# B&R Automation Studio project GroupProjectBR
Automation Studio 4.12.4.107 SP; Project that includes both HMI visualization and script of controling conveyor belt and sorting system.; technology packages: mapp 5.23.0, mappCockpit 5.23.0, mappMotion 5.23.0, mappView 5.23.0, mappVision 5.23.0

## Configuration ConfigSortingSystem

CPU , AutomationRuntime B4.93, Build 4.1.2, Safety 0.0, Vc V4.72.6

### Task classes (Cpu.sw)
```
Cyclic#1 (cycle 8000 us, tolerance 0 us):
  Auto <- Programs.Auto.prg
  Manual <- Programs.Manual.prg
  SemiAuto <- Programs.SemiAuto.prg
Cyclic#3:
  Camera <- Programs.Camera.prg
  ProgramRec <- Programs.RecipesMgmnt.prg
Cyclic#6:
  Alarms <- Programs.Alarms.prg
DataObjects: McAcpSys
NcDataObjects: McDriveLog
Binaries: McAcpDrv, udbdef, McAcpSim, mvLoader, arflatprv, TCLang, visionUnit, mCoWebSc, TCData, FWRules, arcoal, arsvcreg, SettingsVi, sysconf, Settings, iomap, asfw, Role, ashwac, gRecipeXML, Config_2, arconfig, viAppLogo, Config_1, TC, ashwd, Config, User, Config_3, viAppLogoR, viComp4, viComp1, ViApplicat, Config_5, viComp
Libraries: McBase, MpAxis, McAxis, MpBase, McAcpAx, CoTrace, AsZip, FileIO, runtime, ViBase, AsARCfg, powerlnk, MpRecipe, AsEPL, AsIO, DataObj, astime, MpAlarmX, MpServer, standard, AsHttp, asstring, MpUserX, MpFile, asieccon, aruser, arssl, sys_lib, arcert, ashw, aseth, asbrstr, asusb, MpAudit, MpReport
```

### Hardware
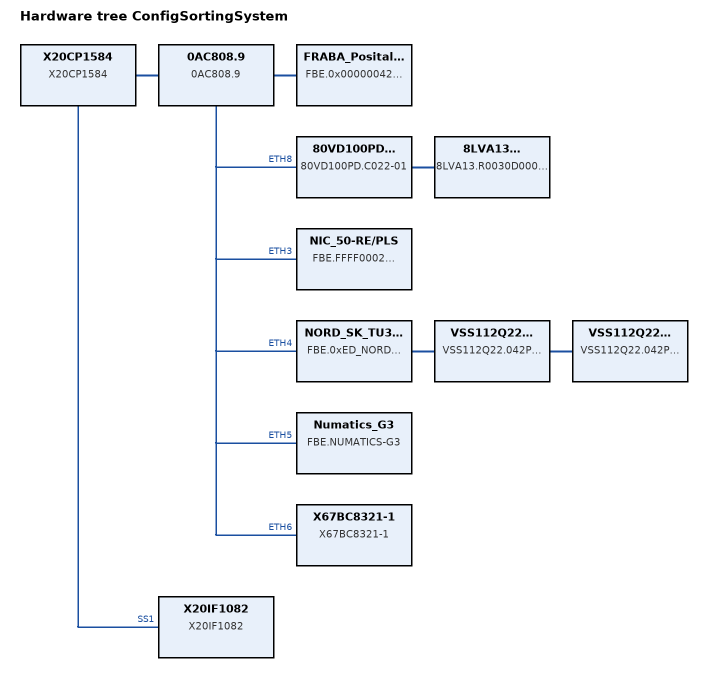
```
0AC808.9 : 0AC808.9 v1.0.0.0  [ETH1 -> X20CP1584.IF3 [Cable Type=PowerlinkCable, Length=10, Version=1.0.0.3]; ETH2 -> FRABA_Posital_Absolute_Rotary_Encoder.PLK1 [Cable Type=PowerlinkCable, Length=10, Version=1.0.0.3]; ETH3 -> NIC_50-RE/PLS.PLK1 [Cable Type=PowerlinkCable, Length=10, Version=1.0.0.3]; ETH4 -> NORD_SK_TU3-POL_SK54xE_Inverter.PLK1 [Cable Type=PowerlinkCable, Length=10, Version=1.0.0.3]; ETH5 -> Numatics_G3.PLK1 [Cable Type=PowerlinkCable, Length=10, Version=1.0.0.3]; ETH6 -> X67BC8321-1.PLK1 [Cable Type=PowerlinkCable, Length=10, Version=1.0.0.3]; ETH8 -> 80VD100PD.C022-01.PLK1 [Cable Type=PowerlinkCable, Length=10, Version=1.0.0.3]]
80VD100PD.C022-01 : 80VD100PD.C022-01 v2.5.0.0  [PLK1 -> 0AC808.9.ETH8 (NodeNumber=9) [Cable Type=PowerlinkCable, Length=10, Version=1.0.0.3]; EC1 -> 8LVA13.R0030D000-0b.EC]
  DriveConfiguration/Module:
    McAcoposTypeID = AcoposMicroDConfig
    ActivateACOPOSSimulationOnPLC = 0
  DriveConfiguration/Encoder/EncoderX6A/InterfaceType:
    ResolverPolepairs = 1
  DriveConfiguration/Encoder/EncoderX6B/InterfaceType:
    ResolverPolepairs = 1
  DriveConfiguration/Channel[1]/RealAxis:
    AxisReference = gAxis_1
    MechanicalElementsIsInvisible = 0
  DriveConfiguration/Channel[1]/RealAxis/MechanicalElements/Gearbox:
    InputIsReadOnly = 0
    Input = 1
    OutputIsReadOnly = 0
    Output = 1
  DriveConfiguration/Channel[1]/RealAxis/MechanicalElements/RotaryToLinearTransformation:
    ReferenceDistanceIsReadOnly = 0
    ReferenceDistance = 175
  DriveConfiguration/Channel[1]/RealAxis/Controller:
    ModeIsReadOnly = 0
    Mode = PositionController
  DriveConfiguration/Channel[1]/RealAxis/Controller/Mode/Position:
    ProportionalGain = 52
    IntegrationTime = 0.0
    PredictionTime = 0.0004
    TotalDelayTime = 0.0004
  DriveConfiguration/Channel[1]/RealAxis/Controller/Mode/Speed:
    ProportionalGainIsReadOnly = 0
    ProportionalGain = 1.1
    IntegrationTimeIsReadOnly = 0
    IntegrationTime = 0.0065
    FilterTimeIsReadOnly = 0
    FilterTime = 0.0
  DriveConfiguration/Channel[1]/RealAxis/Controller/Mode/LoopFilters:
    LoopFilterXIsReadOnly = 0
    LoopFilter1 = Lowpass
  DriveConfiguration/Channel[1]/RealAxis/Controller/Mode/LoopFilters/LoopFilter1:
    CutOffFrequency = 800
  DriveConfiguration/Channel[1]/RealAxis/Controller/Mode/LoopFilters:
    LoopFilter2 = NotUsed
    LoopFilter3 = NotUsed
  DriveConfiguration/Channel[1]/RealAxis/Homing:
    ModeIsReadOnly = 0
    Mode = Direct
  DriveConfiguration/Channel[1]/RealAxis/Homing/Mode:
    Position = 0.0
    ReferencePulse = NotUsed
  DriveConfiguration/Channel[1]/RealAxis/Homing:
    RestorePositionVariable = 
  DriveConfiguration/Channel[1]/RealAxis/StopReaction:
    QuickstopIsReadOnly = 0
    Quickstop = DecelerationLimit
    DriveErrorIsReadOnly = 0
    DriveError = DecelerationLimit
  DriveConfiguration/Channel[1]/RealAxis/MovementErrorLimits:
    PositionError = 5
    VelocityErrorMonitoring = Automatic1
  DriveConfiguration/Channel[1]/RealAxis:
    JerkFilterIsReadOnly = 0
    JerkFilter = NotUsed
    ZeroVibrationFilter = NotUsed
  DriveConfiguration/Channel[1]/RealAxis/DigitalInputs/HomingSwitch:
    SourceIsReadOnly = 0
    Source = NotUsed
    Level = High
  DriveConfiguration/Channel[1]/RealAxis/DigitalInputs/PositiveLimitSwitch:
    SourceIsReadOnly = 0
    Source = NotUsed
    Level = High
  DriveConfiguration/Channel[1]/RealAxis/DigitalInputs/NegativeLimitSwitch:
    SourceIsReadOnly = 0
    Source = NotUsed
    Level = High
  DriveConfiguration/Channel[1]/RealAxis/DigitalInputs/Trigger1:
    Source = X2Trigger1
    Level = High
  DriveConfiguration/Channel[1]/RealAxis/DigitalInputs/Trigger2:
    Source = X2Trigger2
    Level = High
  DriveConfiguration/Channel[1]/RealAxis/DigitalInputs/Quickstop:
    Input = Trigger2
  DriveConfiguration/Channel[1]/RealAxis/Simulation:
    SimulationModeOnPLC = SetValueGeneration
    SimulationModeOnACOPOS = NotUsed
  DriveConfiguration/Channel[2]/RealAxis:
    AxisReference = 
    MechanicalElementsIsInvisible = 0
  DriveConfiguration/Channel[2]/RealAxis/MechanicalElements/Gearbox:
    InputIsReadOnly = 0
    Input = 1
    OutputIsReadOnly = 0
    Output = 1
  DriveConfiguration/Channel[2]/RealAxis/MechanicalElements/RotaryToLinearTransformation:
    ReferenceDistanceIsReadOnly = 0
    ReferenceDistance = 1
  DriveConfiguration/Channel[2]/RealAxis/Controller:
    ModeIsReadOnly = 0
    Mode = PositionController
  DriveConfiguration/Channel[2]/RealAxis/Controller/Mode/Position:
    ProportionalGain = 50.0
    IntegrationTime = 0.0
    PredictionTime = 0.0004
    TotalDelayTime = 0.0004
  DriveConfiguration/Channel[2]/RealAxis/Controller/Mode/Speed:
    ProportionalGainIsReadOnly = 0
    ProportionalGain = 2.0
    IntegrationTimeIsReadOnly = 0
    IntegrationTime = 0.0
    FilterTimeIsReadOnly = 0
    FilterTime = 0.0
  DriveConfiguration/Channel[2]/RealAxis/Controller/Mode/LoopFilters:
    LoopFilterXIsReadOnly = 0
    LoopFilter1 = NotUsed
    LoopFilter2 = NotUsed
    LoopFilter3 = NotUsed
  DriveConfiguration/Channel[2]/RealAxis/Homing:
    ModeIsReadOnly = 0
    Mode = Direct
  DriveConfiguration/Channel[2]/RealAxis/Homing/Mode:
    Position = 0.0
    ReferencePulse = NotUsed
  DriveConfiguration/Channel[2]/RealAxis/Homing:
    RestorePositionVariable = 
  DriveConfiguration/Channel[2]/RealAxis/StopReaction:
    QuickstopIsReadOnly = 0
    Quickstop = DecelerationLimit
    DriveErrorIsReadOnly = 0
    DriveError = DecelerationLimit
  DriveConfiguration/Channel[2]/RealAxis/MovementErrorLimits:
    PositionError = 1.0
    VelocityErrorMonitoring = Automatic1
  DriveConfiguration/Channel[2]/RealAxis:
    JerkFilterIsReadOnly = 0
    JerkFilter = NotUsed
    ZeroVibrationFilter = NotUsed
  DriveConfiguration/Channel[2]/RealAxis/DigitalInputs/HomingSwitch:
    SourceIsReadOnly = 0
    Source = NotUsed
    Level = High
  DriveConfiguration/Channel[2]/RealAxis/DigitalInputs/PositiveLimitSwitch:
    SourceIsReadOnly = 0
    Source = NotUsed
    Level = High
  DriveConfiguration/Channel[2]/RealAxis/DigitalInputs/NegativeLimitSwitch:
    SourceIsReadOnly = 0
    Source = NotUsed
    Level = High
  DriveConfiguration/Channel[2]/RealAxis/DigitalInputs/Trigger1:
    Source = X2Trigger1
    Level = High
  DriveConfiguration/Channel[2]/RealAxis/DigitalInputs/Trigger2:
    Source = X2Trigger2
    Level = High
  DriveConfiguration/Channel[2]/RealAxis/DigitalInputs/Quickstop:
    Input = Trigger2
  DriveConfiguration/Channel[2]/RealAxis/Simulation:
    SimulationModeOnPLC = SetValueGeneration
    SimulationModeOnACOPOS = NotUsed
8LVA13.R0030D000-0b : 8LVA13.R0030D000-0 v2.2.0.4  [EC -> 80VD100PD.C022-01.EC1; MT -> 80VD100PD.C022-01.MT1]
  M1/MotorParameters:
    MOTOR_AMB_TEMP_RATED = 40
FRABA_Posital_Absolute_Rotary_Encoder : FBE.0x00000042_PowerlinkRotaryEncoder_OCD_V02-10 v1.0 (OrderNumber=FRABA Posital Absolute Rotary Encoder)  [PLK1 -> 0AC808.9.ETH2 (NodeNumber=8) [Cable Type=PowerlinkCable, Length=10, Version=1.0.0.3]]
  Supervision = off
  p2110_value = 
  p6000_value = 
  p6003_value = 
NIC_50-RE/PLS : FBE.FFFF0002_TLBPOWERLINK v1.0 (OrderNumber=NIC 50-RE/PLS)  [PLK1 -> 0AC808.9.ETH3 (NodeNumber=2) [Cable Type=PowerlinkCable, Length=10, Version=1.0.0.3]]
  Supervision = off
NORD_SK_TU3-POL_SK54xE_Inverter : FBE.0xED_NORD_TU3_POL_SK54xE_Inverter v1.0 (OrderNumber=NORD SK TU3-POL SK54xE Inverter)  [PLK1 -> 0AC808.9.ETH4 (NodeNumber=3) [Cable Type=PowerlinkCable, Length=10, Version=1.0.0.3]; PLK2 -> VSS112Q22.042P-000.PLK1 (NodeNumber=3) [Cable Type=PowerlinkCable, Length=10, Version=1.0.0.3]]
  Supervision = off
Numatics_G3 : FBE.NUMATICS-G3 v1.0 (OrderNumber=Numatics G3)  [PLK1 -> 0AC808.9.ETH5 (NodeNumber=6) [Cable Type=PowerlinkCable, Length=10, Version=1.0.0.3]]
  Supervision = off
VSS112Q22.042P-000 : VSS112Q22.042P-000 v1.8.0.674  [PLK1 -> NORD_SK_TU3-POL_SK54xE_Inverter.PLK2 (NodeNumber=1) [Cable Type=PowerlinkCable, Length=10, Version=1.0.0.3]; PLK2 -> VSS112Q22.042P-000a.PLK1 (NodeNumber=1) [Cable Type=PowerlinkCable, Length=10, Version=1.0.0.3]]
  Supervision = off
  VisionConfig = gCamera
VSS112Q22.042P-000a : VSS112Q22.042P-000 v1.8.0.674  [PLK1 -> VSS112Q22.042P-000.PLK2 (NodeNumber=12) [Cable Type=PowerlinkCable, Length=10, Version=1.0.0.3]]
  Supervision = off
  VisionConfig = gCamera_C
X20CP1584 : X20CP1584 v1.10.0.0
  Connector IF2:
    ActivateDevice = 1
    Mode = Manual
    InternetAddress = 192.168.0.100
    SubnetMask = 255.255.255.0
    ActivateSnmp = 2
  Connector IF3:
    MtuSize = 1500
    CycleTime = 400
    InternetAddress = 192.168.200.240
    SubnetMask = 255.255.255.0
    ActivateANSL = 1
  ConfigurationID = Group_Project_BR_ConfigSortingSystem
  TimerDeviceType = EPLX2X
  TimerDevice = X20CP1584.IF3
  TaskClassIdleTime = 2000
  Cyclic1Duration = 8000
  Cyclic1Tolerance = 0
  FileDevice1
  FileDeviceName1 = CF
  FileDevicePath1 = F:\Recipes
  FileDevice2
  FileDeviceName2 = CF_A
  FileDevicePath2 = F:\Alarms
  FileDevice3
  FileDeviceName3 = EF
  FileDevicePath3 = F:\
  FileDevice4
  FileDeviceName4 = CF_Au
  FileDevicePath4 = F:\Audit
  TimeZone = 160
  ActivateDaylightSavingTime = 1
  FtpUser1
  FtpUsername1 = admin
  FtpUserPassword1 = WeMTPAcm1nzSLzz2jYHCDrnHk4ZzO0PbajRql3XcDX4=  // admin
  FtpUserSalt1 = 5SVs8NA4
  FTPAccessRight1 = 0
  ActivateOpcUa = 1
  OpcUaActivateAuditEvents = 1
  OpcUa_Security_AdminRole = Administrator
  OpcUaInformationModels_PV_Version = 1
X20IF1082 : X20IF1082 v1.11.0.0  [SS -> X20CP1584.SS1]
  Connector IF1:
    EplNatSubnet = 192.168.102.0
X67BC8321-1 : X67BC8321-1 v2.14.0.0  [PLK1 -> 0AC808.9.ETH6 (NodeNumber=5) [Cable Type=PowerlinkCable, Length=10, Version=1.0.0.3]]
```

### IoMap.iom - X20CP1584/IoMap.iom
```iecst
VAR_CONFIG
	::gInWeightMeasure AT %IB."NIC_50-RE/PLS"._1ByteIn_04_I2100_S04;
	::gActuatorByte AT %QW."Numatics_G3".Out01_I3201Out;
	::Alarms:ModuleOkScale AT %IX."NIC_50-RE/PLS".ModuleOk;
	::Alarms:ModuleOkInverter AT %IX."NORD_SK_TU3-POL_SK54xE_Inverter".ModuleOk;
	::Alarms:ModuleOkPLC_PLK AT %IX."X20IF1082".ModuleOk;
	::Alarms:ModuleOkEncoder AT %IX."FRABA_Posital_Absolute_Rotary_Encoder".ModuleOk;
	::Alarms:ModuleOkActuators AT %IX."Numatics_G3".ModuleOk;
	::Alarms:ModuleOkPneu_X67BC AT %IX."X67BC8321-1".ModuleOk;
	::Camera:Logo.ModuleOK AT %IX."VSS112Q22.042P-000".ModuleOk;
	::Camera:Logo.LED AT %QB."VSS112Q22.042P-000".StatusLED;
	::Camera:Logo.PhotoTaken AT %IB."VSS112Q22.042P-000".CompletedAcquisitionCnt;
	::Camera:Logo.SetFocus AT %QW."VSS112Q22.042P-000".SetFocus;
	::Camera:Logo.SetExpo AT %QD."VSS112Q22.042P-000".ExposureTime01;
	::Camera:Logo.FlashColor AT %QB."VSS112Q22.042P-000".FlashColor01;
	::Camera:Logo.FlashSegments AT %QB."VSS112Q22.042P-000".FlashSegment01;
	::Camera:Logo.ImgProcessingActive AT %IX."VSS112Q22.042P-000".ImageProcessingActive;
	::Camera:Logo.ImageAcq AT %QX."VSS112Q22.042P-000".ImageAcquisition;
	::Camera:Logo.Enable AT %QX."VSS112Q22.042P-000".EnableMatch;
	::Camera:Logo.NumSearchMax AT %QB."VSS112Q22.042P-000".NumSearchMaxMatch;
	::Camera:Logo.MIN_SCORE AT %QB."VSS112Q22.042P-000".MinScoreMatch;
	::Camera:Logo.MAX_OVERLAP AT %QB."VSS112Q22.042P-000".MaxOverlapMatch;
	::Camera:Logo.NumberMatches AT %IB."VSS112Q22.042P-000".NumResultsMatch;
	::Camera:Logo.Model_ID AT %IB."VSS112Q22.042P-000".ModelNumberMatch01;
	::Camera:Logo.MatchScore AT %IB."VSS112Q22.042P-000".ScoreMatch01;
	::Camera:Logo.ReadFocus AT %IW."VSS112Q22.042P-000".ReadFocus;
	::Camera:Logo.ReadExpo AT %ID."VSS112Q22.042P-000".ReadExposureTime;
	::Camera:Color.LED AT %QB."VSS112Q22.042P-000a".StatusLED;
	::Camera:Color.ResultsMatch AT %IB."VSS112Q22.042P-000a".NumResults;
	::Camera:ColorIdModel AT %IB."VSS112Q22.042P-000a".ColorIdModel01;
	::Camera:Color.Model_ID AT %IB."VSS112Q22.042P-000a".ModelNumber01;
	::Camera:Color.Enable AT %QX."VSS112Q22.042P-000a".Enable;
	::Camera:Color.NumSearchMax AT %QB."VSS112Q22.042P-000a".NumSearchMax;
	::Camera:Color.RegionFeatures AT %QX."VSS112Q22.042P-000a".RegionFeatures;
	::Camera:Color.EnhancedBlobInfo AT %QX."VSS112Q22.042P-000a".EnhancedBlobInfo;
	::Camera:Color.Alignment AT %QB."VSS112Q22.042P-000a".Alignment;
	::Camera:Color.SetFocus AT %QW."VSS112Q22.042P-000a".SetFocus;
	::Camera:Color.SetExpo AT %QD."VSS112Q22.042P-000a".ExposureTime01;
	::Camera:Color.FlashColor AT %QB."VSS112Q22.042P-000a".FlashColor01;
	::Camera:Color.FlashSegments AT %QB."VSS112Q22.042P-000a".FlashSegment01;
	::Camera:Color.ImageAcq AT %QX."VSS112Q22.042P-000a".ImageAcquisition;
	::Camera:Color.ModuleOK AT %IX."VSS112Q22.042P-000a".ModuleOk;
	::Auto:ScaleTare AT %QB."NIC_50-RE/PLS"._1ByteOut_02_I2000_S02;
	::Camera:Color.ReadFocus AT %IW."VSS112Q22.042P-000a".ReadFocus;
	::Camera:Color.ReadExpo AT %ID."VSS112Q22.042P-000a".ReadExposureTime;
	::Camera:Color.PhotoTaken AT %IB."VSS112Q22.042P-000a".CompletedAcquisitionCnt;
	::Camera:Color.ImgProcessingActive AT %IX."VSS112Q22.042P-000a".ImageProcessingActive;
END_VAR
```

### Config_1.axis - X20CP1584/mappMotion/Config_1.axis
```
Element gAxis_1 (Type=axis)
  BaseTypeIsReadOnly = 0
  BaseType = Linear
    MeasurementUnit = 5066068
    MeasurementResolutionIsReadOnly = 0
    MeasurementResolution = 0.01
    CountDirectionIsReadOnly = 0
    CountDirection = Standard
  MovementLimitsIsReadOnly = 0
  MovementLimits = Internal
    Position:
      LowerLimitMin = -1.79769313486231E308
      UpperLimitMax = 1.79769313486231E308
      LowerLimit = -1000.0
      UpperLimit = 1000.0
    VelocityIsReadOnly = 0
    Velocity:
      VelocityMax = 3.4E38
      Velocity = 500
    AccelerationIsReadOnly = 0
    Acceleration:
      AccelerationMax = 3.4E38
      Acceleration = 2500
    DecelerationIsReadOnly = 0
    Deceleration:
      DecelerationMax = 3.4E38
      Deceleration = 2500
  Alarms = None
```

### Config.mpalarmxcore - X20CP1584/mappServices/Config.mpalarmxcore
```
Element gAlarmXCore (Type=mpalarmxcore)
  mapp.AlarmX.Core.Configuration:
    [0]:
      Name = Unrecognized object
      Message = Attempt to classify object has failed
      Behavior = DiscreteValueMonitoring
        Monitoring:
          MonitoredPV = ::Auto:State
          TriggerValues:
            [0] = 17
    [1]:
      Name = Left box is full
      Message = Left box reached maximum ammount of objects in it
      Behavior = DiscreteValueMonitoring
        Monitoring:
          MonitoredPV = ::Auto:AlarmLeft
          TriggerValues:
            [0] = 1
    [2]:
      Name = Right box is full
      Message = Right box reached maximum ammount of objects in it
      Behavior = DiscreteValueMonitoring
        Monitoring:
          MonitoredPV = ::Auto:AlarmRight
          TriggerValues:
            [0] = 1
    [3]:
      Name = Motor error
      Message = gMotorBeltAxisBasic has returned an error. Manual restart is required in "Service" page.
      Behavior = DiscreteValueMonitoring
        Monitoring:
          MonitoredPV = ::gMotorBeltAxisBasic.Error
          TriggerValues:
            [0] = 1
    [4]:
      Name = Hardware error
      Message = No connection to at least on module. Fix connections and reset hardware via service page
      Behavior = DiscreteValueMonitoring
        Monitoring:
          MonitoredPV = ::gAlarmHardware
          TriggerValues:
            [0] = 1
```

### Config_3.mpuserx - X20CP1584/mappServices/Config_3.mpuserx
```
Element UserMgmtX (Type=mpuserx)
  ServerSettings:
    Server:
      AdditionalUserData:
        [0] = mail
        [1] = telephoneNumber
  Groups:
    DefGroup#1:
      id = Administrator
      admin = TRUE
    DefGroup#2:
      id = Everyone
      level = 1
    DefGroup#3:
      id = Operator
      level = 3
    DefGroup#4:
      id = Operator
      level = 2
```

### Config_4.mpaudittrail - X20CP1584/mappServices/Config_4.mpaudittrail
```
Element gAuditTrail (Type=mpaudittrail)
  Audit:
    Events:
      [0] = 2
      [1] = 113
      [2] = 48
      [3] = 33
      [4] = 19
    TextSource = TXT
      Name = 
      OutputFormat = Audit/Event/Root
    Archive = On
    Export:
      FileType = 2
      PassPhrase = admin
      PDF:
        UserPassword = 
        Header = 
        Title:
          Text = 
  Monitor:
    0:
      pv = ::Auto:State
  Alarms = MpAlarmX
```

### Config_5.mpfilemanagerui - X20CP1584/mappServices/Config_5.mpfilemanagerui
```
Element gFileManagUI (Type=mpfilemanagerui)
```

### Config_6.mpreportcore - X20CP1584/mappServices/Config_6.mpreportcore
```
Element gReport (Type=mpreportcore)
  MpReport:
    Settings:
      LanguageDependent:
        [0]:
          Language = en
        [1]:
          Language = pl
    PageLayouts:
      [0]:
        Name = Default
    Styles:
      Text:
        [0]:
          Name = Default
      Table:
        [0]:
          Name = Default
      Line:
        [0]:
          Name = Default
      Chart:
        PieChart:
          [0]:
            Name = Default
        LineChart:
          [0]:
            Name = Default
        BarChart:
          [0]:
            Name = Default
    Reports:
      [0]:
        PageLayout = Default
        [0]
  Alarms = MpAlarmX
```

### gRecipeXML.mprecipexml - X20CP1584/mappServices/gRecipeXML.mprecipexml
```
Element gRecipeXml (Type=mprecipexml)
  mapp.Recipe.Xml:
    AutoSave = Time
```

### viComp1.visioncomponent - X20CP1584/mappVision/viComp1.visioncomponent
```
Element gCamera (Type=visioncomponent)
  VisionApplicationReference = viAppLogof
```

### viComp4.visioncomponent - X20CP1584/mappVision/viComp4.visioncomponent
```
Element gCamera_C (Type=visioncomponent)
  VisionApplicationReference = ViApplicationColorful
```

## Logical view

Binary libraries used (declarations not repeated): operator, runtime, astime, AsIecCon, MpAxis 5.23.0, McAxis 5.23.0, MpBase 5.23.0, McAcpAx 5.23.0, CoTrace 5.23.0, AsZip, FileIO, McBase 5.23.0, MpRecipe 5.23.0, asstring, ViBase 5.23.0, AsARCfg, powerlnk, AsEPL, AsIO, DataObj, MpAlarmX 5.23.0, MpServer 5.23.0, standard, AsHttp, MpUserX 5.23.0, MpFile, MpAudit 5.23.0, MpReport 5.23.0

### Global.typ - Global data types
```iecst
TYPE
	ModelEnum :
		(
		BR_Szary := 1, (*%ID of B&R logo model*)
		AS_Oranz := 2, (*%ID of AS logo model*)
		Unrecognised := 0 (*%case of nothing recognised*)
		);
	SortingType : 	STRUCT
		RecipeName : STRING[80];
		Date : STRING[80];
		SortChoice : SortChoiceEnum;
		SortLeftMin : BOOL;
		SortLeftBR : BOOL;
		SortLeftGrey : BOOL;
		ItemWeightLeftMin : USINT;
		ItemWeightLeftMax : USINT;
		ItemWeightRightMin : USINT;
		ItemWeightRightMax : USINT;
		ItemWeightBorderWeight : USINT;
		Threshold : BOOL;
		LeftCriteria : Criteria;
		RightCriteria : Criteria;
	END_STRUCT;
	SortChoiceEnum :
		(
		WEIGHT := 0,
		OPTIC_LOGO := 1,
		OPTIC_COLOR := 2,
		ADVANCED := 3
		);
	Camera_enum_main : 	STRUCT
		ModuleOK : BOOL;
		LED : USINT;
		Model_ID : USINT;
		PhotoTaken : USINT;
		SetFocus : UINT;
		SetExpo : UDINT;
		ReadFocus : UINT;
		ReadExpo : UDINT;
		ImageAcq : BOOL;
		DisplayPhoto : BOOL;
		ImageProcessingActive : BOOL;
	END_STRUCT;
	Criteria : 	STRUCT
		AS : BOOL;
		BR : BOOL;
		Grey : BOOL;
		Orange : BOOL;
		Threshold : BOOL;
		Range : BOOL;
		Heavy : BOOL;
		Light : BOOL;
		WeightMin : USINT;
		WeightMax : USINT;
		WeightBorder : USINT;
	END_STRUCT;
END_TYPE
```

### Global.var - Global variables
```iecst
(*Insert your comment here.*)
VAR
	gActuatorByte : UINT;
	gAddToLeft : BOOL := FALSE;
	gAddToRight : BOOL := FALSE;
	gAlarmExist : BOOL := FALSE;
	gAlarmHardAck : BOOL := FALSE;
	gAlarmHardware : BOOL := FALSE;
	gCTU_QuantityLeft : CTU;
	gCTU_QuantityRight : CTU;
	gCTU_Reset_Left : BOOL := FALSE;
	gCTU_Reset_Right : BOOL := FALSE;
	gErrorState : BOOL := FALSE;
	gInWeightMeasure : USINT;
	gMaxLeftStorage : USINT := 4;
	gMaxRightStorage : USINT := 4;
	gMode : USINT := 0;
	gMotorBeltAxisBasic : MpAxisBasic;
	gMotorBeltParType : MpAxisBasicParType;
	gMpRecipeRegPar_0 : MpRecipeRegPar;
	gMpRecipeUI_0 : MpRecipeUI;
	gMpRecipeXML_0 : MpRecipeXml;
	gPicNotRecognised : BOOL := FALSE;
	gProgCamera : Camera_enum_main := (ImageAcq:=FALSE,DisplayPhoto:=FALSE);
	gQuantityLeftStorage : UINT := 0;
	gQuantityRightStorage : UINT := 0;
	gPhotoShowed : BOOL;
	gRecognisedModel : ModelEnum := Unrecognised;
	gSortChoiceView : BOOL;
	gSorting : SortingType := (RecipeName:='empty',Date:='1970-01-01 01:00:00',SortChoice:=WEIGHT,SortLeftMin:=FALSE,SortLeftBR:=FALSE,SortLeftGrey:=FALSE,ItemWeightLeftMin:=1,ItemWeightLeftMax:=10,ItemWeightRightMin:=11,ItemWeightRightMax:=20,ItemWeightBorderWeight:=10,LeftCriteria:=(WeightMin:=1,WeightMax:=10,WeightBorder:=10),RightCriteria:=(WeightMin:=1,WeightMax:=10,WeightBorder:=10));
	gStopBlink : BOOL := TRUE;
	gStopState : BOOL := TRUE;
	gUIConnect : MpRecipeUIConnectType;
	gUISetup : MpRecipeUISetupType;
	gWeightDetected : BOOL := FALSE;
	gCamera_0L_1C : USINT;
END_VAR
```

### Package Logical/Libraries - Global libraries

- Visualisation Logical/mappView (not shown)

### Program Logical/Programs/Auto (IEC)

#### Types.typ
```iecst
TYPE
	State_ADVANCED :
		(
		WAIT,
		LOGO,
		COLOR,
		THRESHOLD_LEFT,
		THRESHOLD_RIGHT,
		RANGE_LEFT,
		RANGE_RIGHT,
		ADV_WEIGHT
		);
	ProgramStatesEnum :
		(
		STOP := 0,
		INIT := 1,
		START := 2,
		DETECTION := 3,
		CATEGORIZATION := 4,
		TAKE_PICT_CAMERA := 5,
		TAKE_PICT_CAMERA_2 := 6,
		DROP := 7,
		SORT_WEIGHT := 8,
		SORT_OPTIC_LOGO := 9,
		SORT_OPTIC_COLOR := 10,
		SORT_ADVANCED := 11,
		GO_STORAGE_LEFT := 12,
		GO_STORAGE_RIGHT := 13,
		SORT_STORAGE_LEFT := 14,
		SORT_STORAGE_RIGHT := 15,
		UNRECOGNISED_PIC := 16,
		CHOOSE_SORT_MODE := 17,
		DECIDE_WHERE := 18,
		ERROR := 19
		);
END_TYPE
```

#### Variables.var
```iecst
VAR
	ActuatorByte : USINT := 2#0000000000000000;
	ActuatorNotPushing : BOOL;
	ActuatorNotSorting : BOOL;
	ActuatorPushing : BOOL := FALSE;
	ActuatorSorting : BOOL := FALSE;
END_VAR
VAR CONSTANT
	ACTUATOR_BYTE_NOT_ACTIV : USINT := 2#0000000000000000;
	ACTUATOR_BYTE_PUSH : USINT := 2#0000000000000100;
	ACTUATOR_BYTE_SORT : USINT := 2#0000000000000001;
END_VAR
VAR
	HMI_ScaleTare : BOOL := FALSE;
	ItemDetected : BOOL := FALSE;
	ItemWeighLeftMaxBorder : USINT;
	ItemWeighRightMinBorder : USINT;
	ItemWeight : USINT;
	ItemWeightMeasured : USINT;
	MotorHome : BOOL;
	MotorInPosition : BOOL;
	MotorMoveAbsolute : BOOL := FALSE;
	MotorMoveDone : BOOL;
	MotorPos : LREAL;
	MotorPower : BOOL;
	MotorReqAcc : UINT := 700;
	MotorReqDec : UINT := 700;
	MotorReqPosition : UINT := 0;
	MotorReqVel : {REDUND_UNREPLICABLE} UINT := 300;
	MotorVel : REAL;
END_VAR
VAR CONSTANT
	MOTOR_DIST_LEFT : UINT := 90;
	MOTOR_DIST_RIGHT : UINT := 320;
END_VAR
VAR
	NotSelectedAuto : BOOL;
	RESET_ITEM_MEM_WEIGHT : {REDUND_UNREPLICABLE} USINT := 0;
	ScaleTare : USINT := 0;
	SelectedAuto : BOOL;
	ShowBRLeft : BOOL := FALSE;
	ShowBRRight : BOOL := FALSE;
	ShowLightLeft : BOOL := FALSE;
	ShowLightRight : BOOL := FALSE;
	ShowRange : BOOL;
	ShowThreshold : BOOL;
	SortLeftBR_USINT : USINT;
	SortLeftGrey_USINT : USINT;
	SortLeftMin_USINT : USINT;
	Sort_left : BOOL;
	Sort_right : BOOL;
	Start : BOOL := FALSE;
	State : ProgramStatesEnum := STOP;
	State_ADV : State_ADVANCED := WAIT;
	Stop : BOOL := FALSE;
	TimerActuatorOut : BOOL;
	TimerAfterDetect : BOOL;
	TimerCameraPicDone : BOOL;
	TimerTonActuator : TON;
	TimerTonActuatorIn : BOOL := FALSE;
	TimerTonCamera : TON;
	TimerTonDetect : TON;
END_VAR
VAR CONSTANT
	TIME_TON_ACTUATOR : TIME := T#500MS;
	TIME_TON_CAMERA : TIME := T#50ms;
END_VAR
VAR
	TIME_TON_DETECT : TIME := T#2S;
	TIME_TON_SHOW_PHOTO : TIME := T#50ms;
	TimerTONShowPhoto : TON;
	ShowPhoto : BOOL;
	ShowDetectedLabel : BOOL;
	SemiAutoModeSelected : BOOL;
	Approval : BOOL;
	LeftLimit : BOOL;
	RightLimit : BOOL;
	AlarmLeft : BOOL;
	AlarmRight : BOOL;
	Detect : BOOL;
	TooLongDetect : BOOL;
	TimerTooLongDetect : BOOL;
	TON_TooLongDetect : TON;
END_VAR
VAR CONSTANT
	TIME_TON_HOW_LONG_DETECT : TIME := T#2500MS;
END_VAR
```

#### Main.st
```iecst
PROGRAM _INIT

END_PROGRAM

PROGRAM _CYCLIC
	SelectedAuto := (gMode = 0);
	NotSelectedAuto := NOT SelectedAuto;
	SemiAutoModeSelected := (gMode=2);
	// CODE WORKS ONLY WHEN AUTO OR SEMIAUTO IS ACTIVE
	IF  SelectedAuto OR SemiAutoModeSelected THEN

		// MOTOR MANAGEMENT
		gMotorBeltAxisBasic.Enable 		:= TRUE;
		gMotorBeltAxisBasic.MpLink 		:= ADR(gAxis_1);
		gMotorBeltAxisBasic.Parameters 	:= ADR(gMotorBeltParType);
		MotorMoveDone 					:= gMotorBeltAxisBasic.MoveDone;
		gMotorBeltAxisBasic.Power 		:= MotorPower;
		gMotorBeltAxisBasic.Home 		:= MotorHome;
		gMotorBeltAxisBasic();

		// STORAGES OVER LIMIT ACTION
		IF gQuantityLeftStorage >= gMaxLeftStorage THEN
			LeftLimit := TRUE;
		ELSIF gQuantityLeftStorage < gMaxLeftStorage THEN
			LeftLimit := FALSE;
		END_IF;
		IF gQuantityRightStorage >= gMaxRightStorage THEN
			RightLimit := TRUE;
		ELSIF gQuantityRightStorage < gMaxRightStorage THEN
			RightLimit := FALSE;
		END_IF;

		// IN STATE STOP VALUES DOESN'T FLUCTUATE
		IF gMotorBeltAxisBasic.Velocity > 15 THEN
			MotorVel := gMotorBeltAxisBasic.Velocity;
		ELSE
			MotorVel := 0;
		END_IF;
		IF gMotorBeltAxisBasic.Position > 5 THEN
			MotorPos := gMotorBeltAxisBasic.Position;
		ELSE
			MotorPos := 0;
		END_IF;

		// ASSIGNING MOTION PARAMETERS
		gMotorBeltParType.Acceleration 	:= MotorReqAcc;
		gMotorBeltParType.Deceleration 	:= MotorReqDec;
		gMotorBeltParType.Velocity 		:= MotorReqVel;
		gMotorBeltParType.Position 		:= MotorReqPosition;

		// ASSIGNING GLOBAL VARIABLES TO LOCAL VARIABLES
		gActuatorByte					 := ActuatorByte;
		gMotorBeltAxisBasic.Power 		 := MotorPower;
		gMotorBeltAxisBasic.MoveAbsolute := MotorMoveAbsolute;
		gStopState 						 := (State = 0);

		// ASSIGNING LOCAL VARIABLES TO GLOBAL VARIABLES
		MotorInPosition 				 := gMotorBeltAxisBasic.InPosition;
		ItemWeight 						 := gInWeightMeasure;

		// ITEM DETECTION CONDITION
		ItemDetected := (ItemWeight > 1);
		gWeightDetected := ItemDetected;

		// TIMERS
		// actuator
		TimerTonActuator(IN := TimerTonActuatorIn, PT := TIME_TON_ACTUATOR);
		TimerActuatorOut := TimerTonActuator.Q;
		// camera
		TimerTonCamera(IN := gProgCamera.ImageAcq , PT := TIME_TON_CAMERA);
		TimerCameraPicDone := TimerTonCamera.Q;
		// delay after detection
		TimerTonDetect.IN := ItemDetected;
		TimerTonDetect.PT := TIME_TON_DETECT;
		TimerAfterDetect := TimerTonDetect.Q;
		TimerTonDetect();
		// delay after photo
		TimerTONShowPhoto.IN := gProgCamera.ImageAcq;
		TimerTONShowPhoto.PT := TIME_TON_SHOW_PHOTO;
		ShowPhoto := TimerTONShowPhoto.Q;
		TimerTONShowPhoto();
		// timer too long detection
		// delay after photo
		TON_TooLongDetect.IN := TooLongDetect;
		TON_TooLongDetect.PT := TIME_TON_HOW_LONG_DETECT;
		TimerTooLongDetect := TON_TooLongDetect.Q;
		TON_TooLongDetect();

	END_IF;

	// ALARM OR STOP OR AUTO NOT ACTIVE
	IF gAlarmHardware THEN
		IF NOT (State = ERROR) THEN
			State := ERROR;
		END_IF;
	ELSIF Stop OR gMode = 1 OR gAlarmExist THEN
		Stop := FALSE;
		State := STOP;
	END_IF;

	// PROGRAM AUTO
	CASE State OF

		STOP:
			State := STOP;
			IF SelectedAuto OR SemiAutoModeSelected THEN
				MotorPower 		  := FALSE;
				MotorMoveAbsolute := FALSE;
				MotorHome 		  := FALSE;
			END_IF;
			MotorPos := 0;
			MotorVel := 0;
			TimerTonActuatorIn 	  := FALSE;
			ActuatorSorting 	  := FALSE;
			ActuatorPushing  	  := FALSE;
			IF Start THEN
				State := INIT;
			END_IF;

		INIT:
			Sort_left			:= FALSE;
			Sort_right 			:= FALSE;
			gAddToRight 		:= FALSE;
			gAddToLeft 			:= FALSE;
			TimerTonActuatorIn 	:= FALSE;
			ActuatorSorting 	:= FALSE;
			ActuatorPushing 	:= FALSE;
			MotorMoveAbsolute 	:= FALSE;
			MotorPower 			:= TRUE;
			MotorHome 			:= TRUE;
			gPicNotRecognised	:= FALSE;
			Approval 			:= FALSE;
			Detect 				:= FALSE;
			State 				:= START;

		START:
			Approval := FALSE;
			IF ItemDetected THEN
				ItemWeightMeasured 	:= RESET_ITEM_MEM_WEIGHT;
				gRecognisedModel := 0; // NOWE W KODZIE
				State := DETECTION;
			END_IF;

		DETECTION:
			MotorHome 	:= FALSE;
			Approval := FALSE;
			TooLongDetect := TRUE;
			IF TimerAfterDetect THEN
				Detect := TRUE;
				ItemWeightMeasured := ItemWeight;
				State := CATEGORIZATION;
			ELSIF TimerTooLongDetect THEN
				TooLongDetect := FALSE;
				State := START;
			END_IF;

		CATEGORIZATION:
			IF SelectedAuto THEN
				IF gSorting.SortChoice = WEIGHT THEN
					State := CHOOSE_SORT_MODE;
				ELSE
					State := TAKE_PICT_CAMERA;
				END_IF;
			ELSIF SemiAutoModeSelected AND Approval THEN
				IF gSorting.SortChoice = WEIGHT THEN
					Approval := FALSE;
					State := CHOOSE_SORT_MODE;
				ELSE
					Approval := FALSE;
					State := TAKE_PICT_CAMERA;
				END_IF;
			END_IF;

		TAKE_PICT_CAMERA:
			gProgCamera.ImageAcq 	:= TRUE;
			State := TAKE_PICT_CAMERA_2;

		TAKE_PICT_CAMERA_2:
			IF SelectedAuto THEN
				IF NOT gProgCamera.ImageProcessingActive AND TimerCameraPicDone THEN
					gProgCamera.DisplayPhoto := TRUE;
					IF gPhotoShowed THEN
						gPhotoShowed := FALSE;
						IF gRecognisedModel = 0 THEN
							gProgCamera.ImageAcq  := FALSE;
							State 				  := UNRECOGNISED_PIC;
						ELSE
							State 				  := CHOOSE_SORT_MODE;
						END_IF;
					END_IF;
				END_IF;
			ELSIF SemiAutoModeSelected THEN
				IF NOT gProgCamera.ImageProcessingActive AND TimerCameraPicDone THEN
					gProgCamera.DisplayPhoto := TRUE;
					IF gPhotoShowed AND Approval THEN
						gPhotoShowed := FALSE;
						IF gRecognisedModel = 0 THEN
							gProgCamera.ImageAcq  := FALSE;
							Approval := FALSE;
							State 				  := UNRECOGNISED_PIC;
						ELSE
							Approval := FALSE;
							State 				  := CHOOSE_SORT_MODE;
						END_IF;
					END_IF;
				END_IF;
			END_IF;

		CHOOSE_SORT_MODE:
			IF gSorting.SortChoice = OPTIC_LOGO THEN
				State := SORT_OPTIC_LOGO;
			ELSIF gSorting.SortChoice = OPTIC_COLOR THEN
				State := SORT_OPTIC_COLOR;
			ELSIF gSorting.SortChoice = WEIGHT THEN
				State := SORT_WEIGHT;
			ELSIF gSorting.SortChoice = ADVANCED THEN
				State := SORT_ADVANCED;
			END_IF;

			//LONG IF TO PREVENT PROGRAMO KAPUTO
		SORT_WEIGHT:
			IF NOT gSorting.Threshold THEN
				IF (ItemWeightMeasured >= gSorting.ItemWeightLeftMin AND ItemWeightMeasured <= gSorting.ItemWeightLeftMax) AND NOT (ItemWeightMeasured >= gSorting.ItemWeightRightMin AND ItemWeightMeasured <= gSorting.ItemWeightRightMax)  THEN
					IF gSorting.SortLeftMin THEN
						Sort_left := TRUE;
						State := DROP;
					ELSE
						Sort_right := TRUE;
						State := DROP;
					END_IF;
				ELSIF (ItemWeightMeasured >= gSorting.ItemWeightRightMin AND ItemWeightMeasured <= gSorting.ItemWeightRightMax) AND NOT (ItemWeightMeasured >= gSorting.ItemWeightLeftMin AND ItemWeightMeasured <= gSorting.ItemWeightLeftMax) THEN
					IF gSorting.SortLeftMin THEN
						Sort_right := TRUE;
						State := DROP;
					ELSE
						Sort_left := TRUE;
						State := DROP;
					END_IF;
				ELSE
					State := UNRECOGNISED_PIC;
				END_IF;
			ELSE
				IF ItemWeightMeasured < gSorting.ItemWeightBorderWeight THEN
					IF gSorting.SortLeftMin THEN
						Sort_left := TRUE;
						State := DROP;
					ELSE
						Sort_right := TRUE;
						State := DROP;
					END_IF;
				ELSIF ItemWeightMeasured >= gSorting.ItemWeightBorderWeight THEN
					IF gSorting.SortLeftMin THEN
						Sort_right := TRUE;
						State := DROP;
					ELSE
						Sort_left := TRUE;
						State := DROP;
					END_IF;
				END_IF;
			END_IF;

		SORT_OPTIC_LOGO:
			IF gRecognisedModel = 1 THEN
				gProgCamera.ImageAcq 			  := FALSE;					//1
				IF gSorting.SortLeftBR THEN
					Sort_left := TRUE;
					State := DROP;
				ELSE
					Sort_right := TRUE;
					State := DROP;
				END_IF;
			ELSIF gRecognisedModel = 2 THEN
				gProgCamera.ImageAcq 			  := FALSE;						//2
				IF gSorting.SortLeftBR THEN
					Sort_right := TRUE;
					State := DROP;
				ELSE
					Sort_left := TRUE;
					State := DROP;
				END_IF;
			END_IF;

		SORT_OPTIC_COLOR:
			IF gRecognisedModel = 1 THEN
				gProgCamera.ImageAcq 			  := FALSE;						//1
				IF gSorting.SortLeftGrey THEN
					Sort_left := TRUE;
					State := DROP;
				ELSE
					Sort_right := TRUE;
					State := DROP;
				END_IF;
			ELSIF gRecognisedModel = 2 THEN
				gProgCamera.ImageAcq 			  := FALSE;					//2
				IF gSorting.SortLeftGrey THEN
					Sort_right := TRUE;
					State := DROP;
				ELSE
					Sort_left := TRUE;
					State := DROP;
				END_IF;
			END_IF;

		SORT_ADVANCED:
			gProgCamera.ImageAcq  := FALSE;
			CASE State_ADV OF
				WAIT:
					IF gSorting.LeftCriteria.AS OR gSorting.LeftCriteria.BR OR gSorting.RightCriteria.AS OR gSorting.RightCriteria.BR THEN
						State_ADV := LOGO;
					ELSIF gSorting.LeftCriteria.Grey OR gSorting.LeftCriteria.Orange OR gSorting.RightCriteria.Grey OR gSorting.RightCriteria.Orange THEN
						State_ADV := COLOR;
					ELSIF (((gSorting.LeftCriteria.Heavy OR gSorting.LeftCriteria.Light) AND (gSorting.LeftCriteria.Threshold OR gSorting.LeftCriteria.Range)) OR ((gSorting.RightCriteria.Heavy OR gSorting.RightCriteria.Light) AND (gSorting.RightCriteria.Threshold OR gSorting.RightCriteria.Range))) THEN
						State_ADV := ADV_WEIGHT;
					ELSE
						State := UNRECOGNISED_PIC;
					END_IF;

				LOGO:
					//--------------------LEFT----------------------
					IF gSorting.LeftCriteria.BR AND gRecognisedModel = 1 THEN
						IF gSorting.LeftCriteria.Threshold THEN
							State_ADV := THRESHOLD_LEFT;
						ELSIF gSorting.LeftCriteria.Range THEN
							State_ADV := RANGE_LEFT;
						ELSE
							Sort_left := TRUE;
							State := DROP;
						END_IF;
					ELSIF gSorting.LeftCriteria.AS AND gRecognisedModel = 2 THEN
						IF gSorting.LeftCriteria.Threshold THEN
							State_ADV := THRESHOLD_LEFT;
						ELSIF gSorting.LeftCriteria.Range THEN
							State_ADV := RANGE_LEFT;
						ELSE
							Sort_left := TRUE;
							State := DROP;
						END_IF;
						//--------------------RIGHT----------------------
					ELSIF gSorting.RightCriteria.BR AND gRecognisedModel = 1 THEN
						IF gSorting.RightCriteria.Threshold THEN
							State_ADV := THRESHOLD_RIGHT;
						ELSIF gSorting.RightCriteria.Range THEN
							State_ADV := RANGE_RIGHT;
						ELSE
							Sort_right := TRUE;
							State := DROP;
						END_IF;
					ELSIF gSorting.RightCriteria.AS AND gRecognisedModel = 2 THEN
						IF gSorting.RightCriteria.Threshold THEN
							State_ADV := THRESHOLD_RIGHT;
						ELSIF gSorting.RightCriteria.Range THEN
							State_ADV := RANGE_RIGHT;
						ELSE
							Sort_right := TRUE;
							State := DROP;
						END_IF;
					ELSE
						State := UNRECOGNISED_PIC;
					END_IF;

				COLOR:
					//--------------------LEFT----------------------
					IF gSorting.LeftCriteria.Grey AND gRecognisedModel = 1 THEN
						IF gSorting.LeftCriteria.Threshold THEN
							State_ADV := THRESHOLD_LEFT;
						ELSIF gSorting.LeftCriteria.Range THEN
							State_ADV := RANGE_LEFT;
						ELSE
							Sort_left := TRUE;
							State := DROP;
						END_IF;
					ELSIF gSorting.LeftCriteria.Orange AND gRecognisedModel = 2 THEN
						IF gSorting.LeftCriteria.Threshold THEN
							State_ADV := THRESHOLD_LEFT;
						ELSIF gSorting.LeftCriteria.Range THEN
							State_ADV := RANGE_LEFT;
						ELSE
							Sort_left := TRUE;
							State := DROP;
						END_IF;
						//--------------------RIGHT----------------------
					ELSIF gSorting.RightCriteria.Grey AND gRecognisedModel = 1 THEN
						IF gSorting.RightCriteria.Threshold THEN
							State_ADV := THRESHOLD_RIGHT;
						ELSIF gSorting.RightCriteria.Range THEN
							State_ADV := RANGE_RIGHT;
						ELSE
							Sort_right := TRUE;
							State := DROP;
						END_IF;
					ELSIF gSorting.RightCriteria.Orange AND gRecognisedModel = 2 THEN
						IF gSorting.RightCriteria.Threshold THEN
							State_ADV := THRESHOLD_RIGHT;
						ELSIF gSorting.RightCriteria.Range THEN
							State_ADV := RANGE_RIGHT;
						ELSE
							Sort_right := TRUE;
							State := DROP;
						END_IF;
					ELSE
						State := UNRECOGNISED_PIC;
					END_IF;

				ADV_WEIGHT:
					IF gSorting.RightCriteria.Threshold THEN
						State_ADV := THRESHOLD_RIGHT;
					ELSIF gSorting.RightCriteria.Range THEN
						State_ADV := RANGE_RIGHT;
					ELSIF gSorting.LeftCriteria.Threshold THEN
						State_ADV := THRESHOLD_LEFT;
					ELSIF gSorting.LeftCriteria.Range THEN
						State_ADV := RANGE_LEFT;
					END_IF;

				THRESHOLD_LEFT:
					IF ItemWeightMeasured < gSorting.LeftCriteria.WeightBorder THEN
						IF gSorting.LeftCriteria.Light THEN
							Sort_left := TRUE;
							State := DROP;
						ELSE
							State := UNRECOGNISED_PIC;
						END_IF;
					ELSIF ItemWeightMeasured >= gSorting.LeftCriteria.WeightBorder THEN
						IF gSorting.LeftCriteria.Heavy THEN
							Sort_left := TRUE;
							State := DROP;
						ELSE
							State := UNRECOGNISED_PIC;
						END_IF;
					END_IF;

				THRESHOLD_RIGHT:
					IF ItemWeightMeasured < gSorting.RightCriteria.WeightBorder THEN
						IF gSorting.RightCriteria.Light THEN
							Sort_right := TRUE;
							State := DROP;
						ELSE
							State := UNRECOGNISED_PIC;
						END_IF;
					ELSIF ItemWeightMeasured >= gSorting.RightCriteria.WeightBorder THEN
						IF gSorting.RightCriteria.Heavy THEN
							Sort_right := TRUE;
							State := DROP;
						ELSE
							State := UNRECOGNISED_PIC;
						END_IF;
					END_IF;

				RANGE_LEFT:
					IF (ItemWeightMeasured >= gSorting.LeftCriteria.WeightMin AND ItemWeightMeasured <= gSorting.LeftCriteria.WeightMax) THEN
						Sort_left := TRUE;
						State := DROP;
					ELSE
						State := UNRECOGNISED_PIC;
					END_IF;

				RANGE_RIGHT:
					IF (ItemWeightMeasured >= gSorting.RightCriteria.WeightMin AND ItemWeightMeasured <= gSorting.LeftCriteria.WeightMax) THEN
						Sort_right := TRUE;
						State := DROP;
					ELSE
						State := UNRECOGNISED_PIC;
					END_IF;

			END_CASE;

		DROP:
			IF (Sort_left AND LeftLimit) THEN
				AlarmLeft := TRUE;
			ELSIF (Sort_right AND RightLimit) THEN
				AlarmRight := TRUE;
			ELSE
				State_ADV := WAIT;
				ActuatorPushing := TRUE;
				IF SelectedAuto THEN
					IF TimerActuatorOut THEN
						ActuatorPushing := FALSE;
						State := DECIDE_WHERE;
					END_IF;
				ELSIF SemiAutoModeSelected THEN
					IF TimerActuatorOut AND Approval THEN
						ActuatorPushing := FALSE;
						Approval := FALSE;
						State := DECIDE_WHERE;
					END_IF;
				END_IF;
			END_IF;

		DECIDE_WHERE:
			IF Sort_left THEN
				Sort_left := FALSE;
				State := GO_STORAGE_LEFT;
			ELSIF Sort_right THEN
				Sort_right := FALSE;
				State := GO_STORAGE_RIGHT;
			ELSE
				State := UNRECOGNISED_PIC;
			END_IF;

		GO_STORAGE_LEFT:
			IF SelectedAuto THEN
				MotorReqPosition := MOTOR_DIST_LEFT;
				MotorMoveAbsolute := TRUE;
				IF MotorInPosition AND MotorMoveDone THEN
					State := SORT_STORAGE_LEFT;
				END_IF;
			ELSIF SemiAutoModeSelected AND Approval THEN
				MotorReqPosition := MOTOR_DIST_LEFT;
				MotorMoveAbsolute := TRUE;
				IF MotorInPosition AND MotorMoveDone THEN
					Approval := FALSE;
					State := SORT_STORAGE_LEFT;
				END_IF;
			END_IF;

		GO_STORAGE_RIGHT:
			IF SelectedAuto THEN
				MotorReqPosition  := MOTOR_DIST_RIGHT;
				MotorMoveAbsolute := TRUE;
				IF MotorInPosition AND MotorMoveDone THEN
					State := SORT_STORAGE_RIGHT;
				END_IF;
			ELSIF SemiAutoModeSelected AND Approval THEN
				MotorReqPosition  := MOTOR_DIST_RIGHT;
				MotorMoveAbsolute := TRUE;
				IF MotorInPosition AND MotorMoveDone THEN
					Approval := FALSE;
					State := SORT_STORAGE_RIGHT;
				END_IF;
			END_IF;

		SORT_STORAGE_LEFT:
			IF SelectedAuto THEN
				MotorMoveAbsolute := FALSE;
				ActuatorSorting   := TRUE;
				gAddToLeft 		  := TRUE;
				IF TimerActuatorOut THEN
					State := INIT;
				END_IF;
			ELSIF SemiAutoModeSelected THEN
				MotorMoveAbsolute := FALSE;
				IF TimerActuatorOut AND Approval THEN
					Approval := FALSE;
					State := INIT;
				END_IF;
				IF Approval THEN
					ActuatorSorting   := TRUE;
					gAddToLeft 		  := TRUE;
					Approval 		  := FALSE;
				END_IF;
			END_IF;

		SORT_STORAGE_RIGHT:
			IF SelectedAuto THEN
				gAddToRight := TRUE;
				MotorMoveAbsolute := FALSE;
				State := INIT;
			ELSIF SemiAutoModeSelected AND Approval THEN
				Approval := FALSE;
				gAddToRight := TRUE;
				MotorMoveAbsolute := FALSE;
				State := INIT;
			END_IF;

		UNRECOGNISED_PIC:
			State_ADV := WAIT;
			gPicNotRecognised := TRUE;
			State := STOP;

		ERROR:
				MotorPower 		  := FALSE;
				MotorMoveAbsolute := FALSE;
				MotorHome 		  := FALSE;
				MotorPos := 0;
			MotorVel := 0;
			TimerTonActuatorIn 	  := FALSE;
			ActuatorSorting 	  := FALSE;
			ActuatorPushing  	  := FALSE;
			gErrorState := TRUE;
			IF gAlarmHardAck THEN
				IF NOT gAlarmHardware THEN
					gAlarmHardAck := FALSE;
					gErrorState := FALSE;
					State := STOP;
				END_IF;
			END_IF;
	END_CASE;

	// TIMER INPUT TRIGGER TO DELAY ACTUATORS
	IF ActuatorPushing OR ActuatorSorting THEN
		TimerTonActuatorIn := TRUE;
	ELSE
		TimerTonActuatorIn := FALSE;
	END_IF;

	// OPERATION OF BYTE ACTUATORS WITH TIMER
	IF ActuatorPushing THEN
		ActuatorByte := ACTUATOR_BYTE_PUSH;
		IF SelectedAuto THEN
			IF TimerActuatorOut THEN
				ActuatorPushing := FALSE;
			END_IF;
		ELSIF SemiAutoModeSelected THEN
			IF TimerActuatorOut AND Approval THEN
				Approval := FALSE;
				ActuatorPushing := FALSE;
			END_IF;
		END_IF;
	ELSIF ActuatorSorting THEN
		ActuatorByte := ACTUATOR_BYTE_SORT;
		IF SelectedAuto THEN
			IF TimerActuatorOut THEN
				ActuatorSorting := FALSE;
			END_IF;
		ELSIF SemiAutoModeSelected THEN
			IF TimerActuatorOut AND Approval  THEN
				Approval := FALSE;
				ActuatorSorting := FALSE;
			END_IF;
		END_IF;
	ELSE
		ActuatorByte := ACTUATOR_BYTE_NOT_ACTIV;
	END_IF;

	// COUNTERS
	gCTU_QuantityLeft(CU := gAddToLeft, RESET := gCTU_Reset_Left, PV := gMaxLeftStorage);
	gCTU_QuantityRight(CU := gAddToRight, RESET := gCTU_Reset_Right, PV := gMaxRightStorage);
	gQuantityLeftStorage  := gCTU_QuantityLeft.CV;
	gQuantityRightStorage := gCTU_QuantityRight.CV;

	gCTU_QuantityLeft();
	gCTU_QuantityRight();

	IF gCTU_Reset_Left THEN
		AlarmLeft := FALSE;
	END_IF;
	IF gCTU_Reset_Right THEN
		AlarmRight := FALSE;
	END_IF;

	// HMI GUYS WANTED SOME VARIABLES
	IF gSorting.SortChoice <> WEIGHT THEN
		gSortChoiceView := TRUE;
		IF gSorting.SortChoice = ADVANCED THEN
			ShowDetectedLabel := FALSE;
		ELSE
			ShowDetectedLabel := TRUE;
		END_IF;
		ShowLightLeft 	:= FALSE;
		ShowLightRight 	:= FALSE;
		ShowRange 		:= FALSE;
		ShowThreshold 	:= FALSE;
		IF gSorting.SortLeftBR THEN
			ShowBRLeft	:= TRUE;
			ShowBRRight := FALSE;
		ELSE
			ShowBRRight := TRUE;
			ShowBRLeft 	:= FALSE;
		END_IF;
	ELSIF gSorting.SortChoice = WEIGHT THEN
		ShowDetectedLabel := FALSE;
		gSortChoiceView := FALSE;
		ShowBRLeft 		:= FALSE;
		ShowBRRight 	:= FALSE;
		IF gSorting.Threshold THEN
			ShowRange 		:= FALSE;
			ShowThreshold := TRUE;
		ELSE
			ShowRange := TRUE;
			ShowThreshold := FALSE;
		END_IF;

		IF gSorting.SortLeftMin THEN
			ShowLightLeft := TRUE;
			ShowLightRight := FALSE;
		ELSE
			ShowLightRight := TRUE;
			ShowLightLeft := FALSE;
		END_IF;
	END_IF;

	SortLeftMin_USINT := BOOL_TO_USINT(gSorting.SortLeftMin);
	SortLeftBR_USINT := BOOL_TO_USINT(gSorting.SortLeftBR);
	SortLeftGrey_USINT := BOOL_TO_USINT(gSorting.SortLeftGrey);

	//OPC UA - Threshold
	ItemWeighRightMinBorder := gSorting.ItemWeightLeftMax + 1;
	ItemWeighLeftMaxBorder := gSorting.ItemWeightRightMin - 1;

	ActuatorNotSorting := NOT ActuatorSorting;
	ActuatorNotPushing 	:= NOT ActuatorPushing;

	IF Start THEN
		Start := FALSE;
	END_IF;

	//SERVICE PAGE
	//SCALE WEIGHT RESET
	IF HMI_ScaleTare THEN
		ScaleTare := 2#1000;
	ELSE
		ScaleTare := 2#0000;
	END_IF;

END_PROGRAM

PROGRAM _EXIT

END_PROGRAM
```

### Program Logical/Programs/Manual (IEC)

#### Types.typ
```iecst
TYPE
	AxisParam : 	STRUCT
		ManualDistance : LREAL := 500; (*Setting distance of the belt move [mm]*)
		ManualVelocity : REAL := 50; (*Value of velocity [mm/s]*)
	END_STRUCT;
	ManualStepsEnum :
		(
		MANUAL_WAIT := 10,
		MANUAL_BELT_SET_ADDITIVE := 20,
		MANUAL_BELT_MOVE_ADDITIVE := 30,
		MANUAL_BELT_SET_VELOCITY := 40,
		MANUAL_BELT_MOVE_VELOCITY := 50,
		MANUAL_BELT_MOVE_ADDITIVE1 := 60
		);
	ManualStepsActEnum :
		(
		MANUAL_ACTUATOR_WAIT := 200,
		MANUAL_ACTUATOR_DOSING := 210,
		MANUAL_ACTUATOR_NONE := 220,
		MANUAL_ACTUATOR_BOTH := 230,
		MANUAL_ACTUATOR_SORTING := 240
		);
	CameraEnum :
		(
		CAMERA_INIT := 310,
		CAMERA_PHOTO_SHOOT_WAIT := 320,
		CAMERA_PHOTO_DISPLAY_INIT := 330,
		CAMERA_PHOTO_DISPLAY := 340
		);
END_TYPE
```

#### Variables.var
```iecst
VAR
	ImageDisplayTON : TON;
	JogEnableVar : BOOL; (*Jog enablling variable*)
	FlagAdd : BOOL; (*Flag that enables user to see if additive move is active*)
	ManualStep : ManualStepsEnum; (*Enum steps of Manual's state machine*)
	ManualStop : BOOL := FALSE; (*Stopping all of the processes*)
	ManualDistance : LREAL := 300; (*Setting distance of the belt move [mm]*)
	ManualActuatorDosing : BOOL; (*Enabling dosing actuator*)
	ManualActuatorSorting : BOOL; (*Enabling sorting actuator*)
	ManualActuatorBoth : BOOL; (*Enabling both actuators*)
	BeltMoveAdditive : BOOL; (*Activating additive move*)
	ManualActuatorNone : BOOL; (*Disabling both actuators*)
	BeltMoveVelocityOn : BOOL; (*Activating velocity move*)
	BeltMoveVelocityOff : BOOL; (*Disactivating velocity move*)
	ManualVelocity : REAL := 50; (*Value of velocity [mm/s]*)
	DirectionChangeVelocity : BOOL; (*Switching the direction of velocity value / multiplying by -1*)
	DirectionChangeDistance : BOOL; (*Switching the direction of distance value / multiplying by -1*)
	FlagActBoth : BOOL; (*Flag for both enabled actuators*)
	FlagActNone : BOOL; (*Flag for none of enabled actuators*)
	FlagActSorting : BOOL; (*Flag for sorting actuator enabled *)
	FlagActDosing : BOOL; (*Flag for dosing actuator enabled*)
	FlagManual : BOOL; (*Flag that enables user to see if manual mode is enabled*)
	ManualStepAct : ManualStepsActEnum; (*Steps of the actuator state machine*)
	FlagActBothOff : BOOL; (*Flag of the disabled both of actuators*)
	FlagActDosingOff : BOOL; (*Flag of the disabled dosing actuator*)
	FlagActNoneOff : BOOL; (*Flag of the disabled both of actuators*)
	FlagActSortingOff : BOOL; (*Flag of the disabled sorting actuator*)
	FlagNotManual : BOOL; (*Flag that enables user to see if manual mode is disabled*)
	NotMoveActive : BOOL; (*Flag that enables user to see if move is not active*)
	AxisPowerOn : BOOL; (*Enabling power of the motor*)
	FlagArrowLeft : BOOL; (*Motor is rotating to the left side*)
	FlagArrowRight : BOOL; (*Motor is rotating to the right side*)
	AxisPowerOff : BOOL; (*Turning off the power of the axis*)
	FlagVelAddOff : BOOL; (*Flag that enables user to see if additive and velocity move is turned off*)
	PhotoShoot : BOOL; (*Shooting a photo*)
	FlagVel : BOOL; (*Flag that enables user to see if velocity  move is active*)
	sCamera : CameraEnum;
	ImageShootTON : TON;
	MotorVelManual : REAL;
	MotorPosManual : LREAL;
	ShotAvaible : BOOL;
END_VAR
```

#### Main.st
```iecst
PROGRAM _INIT

END_PROGRAM

PROGRAM _CYCLIC

	//-------FUNCTION---BLOCK---CALL-------//
	gMotorBeltAxisBasic();
	ImageShootTON();
	ImageDisplayTON();

	//-------VAR---CALL-------//
	gAxis_1;
	ImageShootTON.PT := T#50ms;
	ImageDisplayTON.PT := T#50ms;

	//----------ALARM----------//
	IF gAlarmHardware THEN								//if module is not ok the error will occour and manual mode will be stopped
		gActuatorByte := 2#0000_0000_0000_0000;
		gMotorBeltAxisBasic.MoveVelocity := 0;
		gMotorBeltAxisBasic.MoveAdditive := 0;
		gMotorBeltAxisBasic.Home := 0;
		gMotorBeltAxisBasic.Power := 0;
	END_IF;

	//--------------DIRECTION---CHANGES--------------//
	IF DirectionChangeVelocity THEN						//changing the direction of the manual distance and manual velocity
		DirectionChangeVelocity := 0;
		ManualVelocity := (-1)*ManualVelocity;
	END_IF;

	IF DirectionChangeDistance THEN
		DirectionChangeDistance := 0;
		ManualDistance := (-1)*ManualDistance;
	END_IF;

	//---------AXIS---VARIABLES---ASSIGMENT----------//

	IF gMode = 1 THEN									//assigning variables value of distance and velocity
		gMotorBeltParType.Distance := ManualDistance;
		gMotorBeltParType.Velocity := ManualVelocity;
		IF gMotorBeltAxisBasic.Velocity > 20 OR gMotorBeltAxisBasic.Velocity < -20 THEN
			MotorVelManual := gMotorBeltAxisBasic.Velocity;
		ELSE
			MotorVelManual := 0;
		END_IF;
		IF gMotorBeltAxisBasic.Position > 5 OR gMotorBeltAxisBasic.Position < -5 THEN
			MotorPosManual := gMotorBeltAxisBasic.Position;
		ELSE
			MotorPosManual := 0;
		END_IF;
	END_IF;

	//-----------------MANUAL---STOP-----------------//
	IF ManualStop THEN									//machine stop
		ManualStop := 0;
		gActuatorByte := 2#0000_0000_0000_0000;
		gMotorBeltAxisBasic.MoveVelocity := 0;
		gMotorBeltAxisBasic.MoveAdditive := 0;
		gMotorBeltAxisBasic.Home := 0;
		gMotorBeltAxisBasic.Power := 0;
		ManualStep := MANUAL_WAIT;
		ManualStepAct := MANUAL_ACTUATOR_WAIT;
	END_IF;

	//----------------------MANUAL---MODE---CHECK---CONDITION----------------------//
	IF (gMode = 1) THEN

		//----------------------STATE---MACHINE---AXIS------------------------//
		CASE ManualStep OF

			MANUAL_WAIT:
				FlagVelAddOff := 1;
				FlagAdd := 0;
				FlagVel := 0;
				IF BeltMoveAdditive THEN				//choosing between axis movement modes; additive
					gMotorBeltAxisBasic.Home := 0;
					BeltMoveAdditive := 0;
					FlagVelAddOff := 0;
					FlagAdd := 1;
					ManualStep := MANUAL_BELT_SET_ADDITIVE;
				ELSIF BeltMoveVelocityOn THEN			//velocity
					gMotorBeltAxisBasic.Home := 0;
					BeltMoveVelocityOn := 0;
					FlagVelAddOff := 0;
					FlagVel := 1;
					ManualStep := MANUAL_BELT_SET_VELOCITY;
				END_IF;

			MANUAL_BELT_SET_ADDITIVE:
				ManualVelocity := ABS(ManualVelocity);	//to avoid error: velocity and distance cannot have a negative value at the same time)
				IF gMotorBeltAxisBasic.PowerOn THEN
					gMotorBeltAxisBasic.Home := 0;
					ManualStep := MANUAL_BELT_MOVE_ADDITIVE;
				END_IF;

			MANUAL_BELT_MOVE_ADDITIVE:
				gMotorBeltAxisBasic.MoveAdditive := 1;
				IF gMotorBeltAxisBasic.MoveDone THEN
					gMotorBeltAxisBasic.ErrorReset := 1;
					gMotorBeltAxisBasic.MoveAdditive := 0;
					ManualStep := MANUAL_BELT_MOVE_ADDITIVE1;
				END_IF;

			MANUAL_BELT_MOVE_ADDITIVE1:
				gMotorBeltAxisBasic.ErrorReset := 0;
				ManualStep := MANUAL_WAIT;

			MANUAL_BELT_SET_VELOCITY:
				IF gMotorBeltAxisBasic.PowerOn THEN
					gMotorBeltAxisBasic.MoveVelocity := 1;
					ManualStep := MANUAL_BELT_MOVE_VELOCITY;
				END_IF;

			MANUAL_BELT_MOVE_VELOCITY:
				IF gMotorBeltAxisBasic.InVelocity THEN
					IF BeltMoveVelocityOff THEN
						BeltMoveVelocityOff := 0;
						gMotorBeltAxisBasic.MoveVelocity := 0;
						ManualStep := MANUAL_WAIT;
					END_IF;
				END_IF;

		END_CASE;

		//-------------------STATE---MACHINE---ACTUATORS---------------------//
		CASE ManualStepAct OF
			MANUAL_ACTUATOR_WAIT:
				IF ManualActuatorDosing THEN					//monostable button for dosing actuator
					ManualActuatorDosing := 0;
					ManualStepAct := MANUAL_ACTUATOR_DOSING;
				ELSIF ManualActuatorSorting THEN				//monostable button for sorting actuator
					ManualActuatorSorting := 0;
					ManualStepAct := MANUAL_ACTUATOR_SORTING;
				ELSIF ManualActuatorBoth THEN					//monostable button for both actuators
					ManualActuatorBoth := 0;
					ManualStepAct := MANUAL_ACTUATOR_BOTH;
				ELSIF ManualActuatorNone THEN					//monostable button for dosing actuator
					ManualActuatorNone := 0;
					ManualStepAct := MANUAL_ACTUATOR_NONE;
				END_IF;

				//actuating actuator responsibile for DOSING an element
			MANUAL_ACTUATOR_DOSING:
				gActuatorByte := 2#0000_0000_0000_0000;
				gActuatorByte := 2#0000_0000_0000_0100;
				ManualStepAct := MANUAL_ACTUATOR_WAIT;

				//actuating actuator responsibile for sorting an element
			MANUAL_ACTUATOR_SORTING:
				gActuatorByte := 2#0000_0000_0000_0000;
				gActuatorByte := 2#0000_0000_0000_0001;
				ManualStepAct := MANUAL_ACTUATOR_WAIT;

				//actuating both actuators
			MANUAL_ACTUATOR_BOTH:
				gActuatorByte := 2#0000_0000_0000_0000;
				gActuatorByte := 2#0000_0000_0000_0101;
				ManualStepAct := MANUAL_ACTUATOR_WAIT;

				//disactuating both actuators
			MANUAL_ACTUATOR_NONE:
				gActuatorByte := 2#0000_0000_0000_0000;
				ManualStepAct := MANUAL_ACTUATOR_WAIT;

		END_CASE;

		//------------END---OF---STATE---MACHINE---ACTUATORS---------------//

		IF AxisPowerOn THEN 											//monostable button enabling axis
			AxisPowerOn := 0;
			gMotorBeltAxisBasic.Power :=1;								//Axis power off is enabling by the button that is binded with stop step
		END_IF;

		IF gMotorBeltAxisBasic.PowerOn THEN			//flag for visualisation purposes
			JogEnableVar := 1;
		ELSE
			JogEnableVar := 0;
		END_IF;

		//------------PHOTO---FUNCTIONS---------------//
		CASE sCamera OF
			CAMERA_INIT:
				ImageShootTON.IN := 0;
				sCamera := CAMERA_PHOTO_SHOOT_WAIT;
				ShotAvaible := TRUE;
			CAMERA_PHOTO_SHOOT_WAIT:
				IF PhotoShoot THEN
					ShotAvaible := FALSE;
					PhotoShoot :=0;
					gProgCamera.ImageAcq 	:= 1;
					sCamera := CAMERA_PHOTO_DISPLAY_INIT;
				END_IF;
			CAMERA_PHOTO_DISPLAY_INIT:
				ImageShootTON.IN := 1;
				IF ImageShootTON.Q THEN
					ImageShootTON.IN := 0;
					gProgCamera.ImageAcq 	:= 0;
					sCamera := CAMERA_PHOTO_DISPLAY;
				END_IF;
			CAMERA_PHOTO_DISPLAY:
				ImageDisplayTON.IN := 1;
				IF ImageDisplayTON.Q THEN
					gProgCamera.DisplayPhoto := TRUE;
					IF gPhotoShowed THEN
						ImageDisplayTON.IN := 0;
						gProgCamera.ImageAcq 	:= 0;
						sCamera := CAMERA_INIT;
					END_IF;
				END_IF;
		END_CASE;

	END_IF;

	//----------------------------FLAG---SECTION----------------------------//
	IF (FlagActDosing = FALSE AND FlagActDosingOff = FALSE) THEN 	//if the power of the axis is enabled
		FlagActDosingOff := TRUE;
	END_IF;

	IF (FlagActSorting = FALSE AND FlagActSortingOff = FALSE) THEN	//if the power of the axis is enabled
		FlagActSortingOff := TRUE;
	END_IF;

	IF gMotorBeltAxisBasic.PowerOn THEN								//if the power of the axis is enabled
		AxisPowerOff := 1;
	ELSE
		AxisPowerOff := 0;
	END_IF;

	IF gMode = 1 THEN												//flag for manual mode choosen
		FlagManual := 1;
		FlagNotManual := 0;
	ELSE
		FlagNotManual := 1;
		FlagManual := 0;
	END_IF;

	IF ManualStepAct = MANUAL_ACTUATOR_DOSING THEN					//flag for dosing actuator
		FlagActBoth := 0;
		FlagActBothOff := NOT(FlagActBoth);
		FlagActDosing := 1;
		FlagActDosingOff := NOT(FlagActDosing);
		FlagActNone := 0;
		FlagActNoneOff := NOT(FlagActNone);
		FlagActSorting := 0;
		FlagActSortingOff := NOT(FlagActSorting);
	ELSIF ManualStepAct = MANUAL_ACTUATOR_SORTING THEN				//flag for sorting actuator
		FlagActBoth := 0;
		FlagActBothOff := NOT(FlagActBoth);
		FlagActDosing := 0;
		FlagActDosingOff := NOT(FlagActDosing);
		FlagActNone := 0;
		FlagActNoneOff := NOT(FlagActNone);
		FlagActSorting := 1;
		FlagActSortingOff := NOT(FlagActSorting);
	ELSIF ManualStepAct = MANUAL_ACTUATOR_BOTH THEN					//flag for both actuators
		FlagActBoth := 1;
		FlagActBothOff := NOT(FlagActBoth);
		FlagActDosing := 1;
		FlagActDosingOff := NOT(FlagActDosing);
		FlagActNone := 0;
		FlagActNoneOff := NOT(FlagActNone);
		FlagActSorting := 1;
		FlagActSortingOff := NOT(FlagActSorting);
	ELSIF ManualStepAct = MANUAL_ACTUATOR_NONE THEN					//flag for none of actuators
		FlagActBoth := 0;
		FlagActBothOff := NOT(FlagActBoth);
		FlagActDosing := 0;
		FlagActDosingOff := NOT(FlagActDosing);
		FlagActNone := 1;
		FlagActNoneOff := NOT(FlagActNone);
		FlagActSorting := 0;
		FlagActSortingOff := NOT(FlagActSorting);
	END_IF;

	IF (((gMotorBeltParType.Distance < 0) AND gMotorBeltAxisBasic.MoveActive AND FlagAdd) OR ((gMotorBeltParType.Velocity <0) AND gMotorBeltAxisBasic.MoveActive AND FlagVel)) THEN		//flag for visibility of left arrow
		FlagArrowLeft := 1;
		FlagArrowRight := 0;
	ELSIF (((gMotorBeltParType.Distance > 0) AND gMotorBeltAxisBasic.MoveActive AND FlagAdd) OR ((gMotorBeltParType.Velocity > 0) AND gMotorBeltAxisBasic.MoveActive AND FlagVel)) THEN	//flag for visibility of right arrow
		FlagArrowRight := 1;
		FlagArrowLeft := 0;
	ELSE								//flag for visibility of none of arrows
		FlagArrowRight := 0;
		FlagArrowLeft := 0;
	END_IF;

	NotMoveActive := NOT(gMotorBeltAxisBasic.MoveActive);
	//----------------------END---OF---FLAG---SECTION----------------------------//

END_PROGRAM

PROGRAM _EXIT

END_PROGRAM
```

### Program Logical/Programs/RecipesMgmnt (IEC)

#### Variables.var
```iecst
VAR
	ClearAudit : BOOL;
	FileLastModified : ARRAY[0..49] OF DATE_AND_TIME;
	idx : INT;
	Filter_sort_type : INT;
	MpAuditTrail_0 : MpAuditTrail;
	MpAuditTrailUI_0 : MpAuditTrailUI;
	AuditUIConnect : MpAuditTrailUIConnectType;
	AuditUISetup : MpAuditTrailUISetupType;
	MpFileManagerUI_0 : MpFileManagerUI;
	FileUIConnect : MpFileManagerUIConnectType;
	FileUISetup : MpFileManagerUISetupType;
	CLEAR_RECIPE : SortingType := (RecipeName:='empty',Date:='1970-01-01 01:00:00',SortChoice:=WEIGHT,SortLeftMin:=TRUE,SortLeftBR:=TRUE,SortLeftGrey:=TRUE,ItemWeightLeftMin:=1,ItemWeightLeftMax:=10,ItemWeightRightMin:=11,ItemWeightRightMax:=20,ItemWeightBorderWeight:=10,Threshold:=TRUE,LeftCriteria:=(AS:=FALSE,BR:=FALSE,Grey:=FALSE,Orange:=FALSE,Threshold:=FALSE,Range:=FALSE,Heavy:=FALSE,Light:=FALSE,WeightMin:=1,WeightMax:=10,WeightBorder:=10),RightCriteria:=(AS:=FALSE,BR:=FALSE,Grey:=FALSE,Orange:=FALSE,Threshold:=FALSE,Range:=FALSE,Heavy:=FALSE,Light:=FALSE,WeightMin:=1,WeightMax:=10,WeightBorder:=10));
END_VAR
VAR RETAIN
	gContainer : ARRAY[0..49] OF SortingType;
END_VAR
VAR
	CurrentFile : STRING[80];
	FileName : ARRAY[0..49] OF STRING[80];
	i : UDINT;
	FileSize : ARRAY[0..49] OF UDINT;
	g : UINT;
	z : UINT;
	Save_Activ : BOOL;
	Clear_param : BOOL;
	CLEAR_ADV_RECIPE : SortingType := (SortChoice:=ADVANCED,SortLeftMin:=FALSE,SortLeftBR:=FALSE,SortLeftGrey:=FALSE,ItemWeightLeftMin:=1,ItemWeightLeftMax:=10,ItemWeightRightMin:=11,ItemWeightRightMax:=20,ItemWeightBorderWeight:=10,Threshold:=FALSE,LeftCriteria:=(AS:=FALSE,BR:=FALSE,Grey:=FALSE,Orange:=FALSE,Threshold:=FALSE,Range:=FALSE,Heavy:=FALSE,Light:=FALSE,WeightMin:=1,WeightMax:=10,WeightBorder:=10),RightCriteria:=(AS:=FALSE,BR:=FALSE,Grey:=FALSE,Orange:=FALSE,Threshold:=FALSE,Range:=FALSE,Heavy:=FALSE,Light:=FALSE,WeightMin:=1,WeightMax:=10,WeightBorder:=10));
	Export_SUCC : BOOL;
	AS_visible : BOOL;
	BR_visible : BOOL;
	Orange_visible : BOOL;
	Grey_visible : BOOL;
	Light_visible : BOOL;
	Heavy_visible : BOOL;
END_VAR
```

#### Main.st
```iecst
PROGRAM _INIT
// ==========================================================================================
// ====================PROGRAM WYMAGA UTWORZENIA 3 FOLDERÓW NA KARCIE PLC!!!=================
// =============Nazwy=Folderów====Audit====Recipes====Alarms=================================
// ==========================================================================================
END_PROGRAM

PROGRAM _CYCLIC
	// AUDIT
	MpAuditTrailUI_0(MpLink := ADR(gAuditTrail), Enable := TRUE, UISetup := AuditUISetup, UIConnect := ADR(AuditUIConnect) );
	MpAuditTrail_0(MpLink := ADR(gAuditTrail), Enable := TRUE, DeviceName := ADR('CF_Au'));
	IF ClearAudit THEN
		MpAuditClearBuffer(MpLink := gAuditTrail);
	END_IF;

	// FILE MANAGEMENT
	MpFileManagerUI_0(MpLink := ADR(gFileManageUI), Enable := TRUE , UISetup := FileUISetup, UIConnect := ADR(FileUIConnect) );
	FileUIConnect.DeviceList.DeviceNames[0] := 'EF';
	i := 0;
	FOR i := 0 TO 15 DO
		FileName[i] := FileUIConnect.File.List.Items[i].Name;
		FileLastModified[i] := FileUIConnect.File.List.Items[i].LastModified;
		FileSize[i] := FileUIConnect.File.List.Items[i].Size;
	END_FOR;

	FileUIConnect.File.List.Items[idx].IsSelected := TRUE;
	CurrentFile := FileUIConnect.File.List.Items[idx].Name;

	CASE Filter_sort_type OF
		0:
			FileUIConnect.File.SortOrder := mpFILE_SORT_BY_NAME_ASC;
		1:
			FileUIConnect.File.SortOrder := mpFILE_SORT_BY_NAME_DESC;
		2:
			FileUIConnect.File.SortOrder := mpFILE_SORT_BY_SIZE_ASC;
		3:
			FileUIConnect.File.SortOrder := mpFILE_SORT_BY_SIZE_DES;
		4:
			FileUIConnect.File.SortOrder := mpFILE_SORT_BY_MOD_TIME_ASC;
		5:
			FileUIConnect.File.SortOrder := mpFILE_SORT_BY_MOD_TIME_DESC;
	END_CASE;

	gMpRecipeRegPar_0.MpLink := 	ADR(gRecipeXml);
	gMpRecipeRegPar_0.Enable :=		TRUE;
	gMpRecipeRegPar_0.PVName := 	ADR('gSorting');

	gMpRecipeXML_0.MpLink := 		ADR(gRecipeXml);
	gMpRecipeXML_0.Enable := 		TRUE;
	gMpRecipeXML_0.DeviceName :=	ADR('CF');

	gMpRecipeUI_0.MpLink :=			ADR(gRecipeXml);
	gMpRecipeUI_0.Enable := 		TRUE;
	gMpRecipeUI_0.UISetup := 		gUISetup;
	gMpRecipeUI_0.UIConnect := 		ADR(gUIConnect);
	gUIConnect.Recipe.SortOrder := mpRECIPE_UI_SORT_DATE_ASCENDING;

	gMpRecipeRegPar_0();
	gMpRecipeXML_0();
	gMpRecipeUI_0();

	IF Clear_param THEN
		gSorting := CLEAR_ADV_RECIPE;
		Clear_param := FALSE;
	END_IF;

	//-----------management-of-adv-buttons--- (almost -30 bindings)
	IF gSorting.LeftCriteria.AS OR gSorting.RightCriteria.AS OR gCamera_0L_1C = 1 THEN
		AS_visible := FALSE;
	ELSE
		AS_visible := TRUE;
	END_IF;
	IF gSorting.LeftCriteria.BR OR gSorting.RightCriteria.BR OR gCamera_0L_1C = 1 THEN
		BR_visible := FALSE;
	ELSE
		BR_visible := TRUE;
	END_IF;
	IF gSorting.LeftCriteria.Orange OR gSorting.RightCriteria.Orange OR gCamera_0L_1C = 0 THEN
		Orange_visible := FALSE;
	ELSE
		Orange_visible := TRUE;
	END_IF;

	IF gSorting.LeftCriteria.Grey OR gSorting.RightCriteria.Grey OR gCamera_0L_1C = 0 THEN
		Grey_visible := FALSE;
	ELSE
		Grey_visible := TRUE;
	END_IF;
	IF gSorting.LeftCriteria.Light OR gSorting.RightCriteria.Light THEN
		Light_visible := FALSE;
	ELSE
		Light_visible := TRUE;
	END_IF;
	IF gSorting.LeftCriteria.Heavy OR gSorting.RightCriteria.Heavy THEN
		Heavy_visible := FALSE;
	ELSE
		Heavy_visible := TRUE;
	END_IF;

END_PROGRAM

PROGRAM _EXIT

END_PROGRAM
```

### Program Logical/Programs/Camera (IEC)

#### Types.typ
```iecst
TYPE
	Camera_enum_color : 	STRUCT
		LED : USINT;
		ModuleOK : BOOL;
		Enable : BOOL;
		NumSearchMax : USINT;
		RegionFeatures : BOOL;
		EnhancedBlobInfo : BOOL;
		Alignment : USINT;
		ImageAcq : BOOL;
		FlashColor : USINT;
		FlashSegments : USINT;
		SetFocus : UINT;
		SetExpo : UDINT;
		ReadFocus : UINT;
		ReadExpo : UDINT;
		Model_ID : USINT;
		ResultsMatch : USINT;
		PhotoTaken : USINT;
		ImgProcessingActive : BOOL;
	END_STRUCT;
	Camera_enum_logo : 	STRUCT
		ModuleOK : BOOL;
		LED : USINT;
		PhotoTaken : USINT;
		ReadFocus : UINT;
		ReadExpo : UDINT;
		SetFocus : UINT;
		SetExpo : UDINT;
		FlashColor : USINT;
		FlashSegments : USINT;
		ImgProcessingActive : BOOL;
		ImageAcq : BOOL;
		Enable : BOOL;
		NumSearchMax : USINT;
		MIN_SCORE : USINT;
		MAX_OVERLAP : USINT;
		NumberMatches : USINT;
		Model_ID : USINT;
		MatchScore : USINT;
	END_STRUCT;
END_TYPE
```

#### Variables.var
```iecst
VAR
	ATON1 : TON;
	ATON2 : TON;
	ATON3 : TON;
	Base64Buffer : STRING[150000];
	Base64srcLen : UDINT;
	CameraLED : USINT := 0;
	CameraLED_2 : USINT := 0;
	httpEncodeBase64_0 : httpEncodeBase64;
END_VAR
VAR CONSTANT
	LED_BLUE : USINT := 4;
END_VAR
VAR
	Logo : Camera_enum_logo := (SetFocus:=17500,SetExpo:=15000,FlashColor:=1,FlashSegments:=1,Enable:=TRUE,NumSearchMax:=1,MIN_SCORE:=44,MAX_OVERLAP:=0);
	Color : Camera_enum_color := (Enable:=TRUE,NumSearchMax:=1,RegionFeatures:=FALSE,EnhancedBlobInfo:=FALSE,Alignment:=0,FlashColor:=1,FlashSegments:=2#0100,SetFocus:=17500,SetExpo:=3000);
END_VAR
VAR CONSTANT
	LED_GREEN : USINT := 2;
	LED_NOTHING : USINT := 1;
	LED_PLC_STATUS : USINT := 0;
	LED_RED : USINT := 3;
END_VAR
VAR
	ManualLampTest : BOOL;
	NewEncodeReq : BOOL;
	sStep : INT;
	TimerTonCameraLED : TON;
	ImageProcess : USINT := 0;
	TimerTonCameraLED_2 : TON;
END_VAR
VAR CONSTANT
	TIMER_TIME_BLINK_100MS : TIME := T#100MS;
	TIMER_TIME_BLINK_500MS : TIME := T#500MS;
	TIME_LAMP_TEST : TIME := T#500MS;
END_VAR
VAR
	URL : STRING[150000];
	URLLength : UDINT;
	ViBaseBuffer : ARRAY[0..150000] OF USINT := [150001(1)];
	ViBaseGetImage_0 : ViBaseGetImage;
	VIBASE_GETIMG_QUALITY : USINT := 40;
	oldFocus : UINT;
	oldExpo : UDINT;
	oldFocusColor : UINT;
	oldExpoColor : UDINT;
	CameraMode : STRING[80];
	Camera_LOGO : BOOL;
	Camera_COLOR : BOOL;
END_VAR
```

#### Main.st
```iecst
PROGRAM _INIT
	//init variables for displaying taken photo in HMI visualization
	URL := '<image x=$'0$' y=$'0$' width=$'320px$' height=$'256px$' href=$'data:application/octet-stream;base64,';
END_PROGRAM

PROGRAM _CYCLIC
	//asfe
	LED_GREEN; //not used, just for some changes
	// MANAGEMENT OF MODE IN CHEAP CAMERA (NO OTHER WAY TO DO THAT :)) )
	IF Logo.ModuleOK THEN
		CameraMode := 'Logo';
		gCamera_0L_1C := 0;
		IF gProgCamera.SetFocus <> oldFocus  THEN
			Logo.SetFocus := gProgCamera.SetFocus;
		END_IF;
		IF gProgCamera.SetExpo <> oldExpo THEN
			Logo.SetExpo := gProgCamera.SetExpo;
		END_IF;
		oldFocus := gProgCamera.SetFocus;
		oldExpo := gProgCamera.SetExpo;

		gProgCamera.ReadExpo := Logo.ReadExpo;
		gProgCamera.ReadFocus := Logo.ReadFocus;

		Logo.LED := gProgCamera.LED;
		Logo.ImageAcq := gProgCamera.ImageAcq;
		gProgCamera.ModuleOK := Logo.ModuleOK;
		gProgCamera.PhotoTaken := Logo.PhotoTaken;
		gProgCamera.Model_ID := Logo.Model_ID;
		gProgCamera.ImageProcessingActive := Logo.ImgProcessingActive;
	ELSIF Color.ModuleOK THEN
		CameraMode := 'Color';
		gCamera_0L_1C := 1;
		IF gProgCamera.SetFocus <> oldFocusColor  THEN
			Color.SetFocus := gProgCamera.SetFocus;
		END_IF;
		IF gProgCamera.SetExpo <> oldExpoColor THEN
			Color.SetExpo := gProgCamera.SetExpo;
		END_IF;
		oldFocusColor := gProgCamera.SetFocus;
		oldExpoColor := gProgCamera.SetExpo;

		gProgCamera.ReadExpo := Color.ReadExpo;
		gProgCamera.ReadFocus := Color.ReadFocus;

		Color.LED := gProgCamera.LED;
		Color.ImageAcq := gProgCamera.ImageAcq;
		gProgCamera.ModuleOK := Color.ModuleOK;
		gProgCamera.PhotoTaken := Color.PhotoTaken;
		gRecognisedModel := Color.Model_ID;
		gProgCamera.Model_ID := Color.Model_ID;
		gProgCamera.ImageProcessingActive := Color.ImgProcessingActive;
	END_IF;

	//-------------CAMERA LED--Blinking-Auto-And-Semiauto-----------//
	//0 - PLC State
	//1 - Nothing
	//2 - Green
	//3 - Red
	//4 - Blue

	IF gMode <> 1 THEN
		IF gAlarmHardware AND NOT gAlarmHardAck THEN
			gStopBlink := FALSE;
			TimerTonCameraLED.PT := TIMER_TIME_BLINK_100MS;
			TimerTonCameraLED_2.PT := TIMER_TIME_BLINK_100MS;
			CameraLED 	:= LED_RED;
			CameraLED_2 := LED_NOTHING;
		ELSIF gAlarmExist THEN
			gStopBlink := FALSE;
			TimerTonCameraLED.PT := TIMER_TIME_BLINK_500MS;
			TimerTonCameraLED_2.PT := TIMER_TIME_BLINK_500MS;
			CameraLED 	:= LED_RED;
			CameraLED_2 := LED_NOTHING;
		ELSIF gPicNotRecognised THEN
			gStopBlink := FALSE;
			TimerTonCameraLED.PT := TIMER_TIME_BLINK_500MS;
			TimerTonCameraLED_2.PT := TIMER_TIME_BLINK_500MS;
			CameraLED 	:= LED_BLUE;
			CameraLED_2 := LED_NOTHING;
		ELSIF gWeightDetected AND NOT gStopState AND NOT gErrorState THEN
			TimerTonCameraLED.PT := TIMER_TIME_BLINK_500MS;
			TimerTonCameraLED_2.PT := TIMER_TIME_BLINK_500MS;
			gStopBlink := FALSE;
			CameraLED 	:= LED_RED;
			CameraLED_2 := LED_BLUE;
		ELSE
			gStopBlink := TRUE;
		END_IF;
	ELSE
		gStopBlink := TRUE;
	END_IF;

	IF gStopBlink THEN
		gProgCamera.LED   := LED_PLC_STATUS;
	ELSE
		TimerTonCameraLED.IN := TRUE;
		gProgCamera.LED := CameraLED;
		IF TimerTonCameraLED.Q THEN
			TimerTonCameraLED_2.IN := TRUE;
			gProgCamera.LED := CameraLED_2;
			IF TimerTonCameraLED_2.Q THEN
				TimerTonCameraLED.IN := FALSE; 				//1 TIMER
				TimerTonCameraLED_2.IN := FALSE;			//2 TIMER
			END_IF;
		END_IF;
	END_IF;

	TimerTonCameraLED();
	TimerTonCameraLED_2();

	//-----------------TEST--CAMERA--LIGHT--------------------//

	ATON1();
	ATON2();
	ATON3();
	IF gMode = 1 THEN
		CASE sStep OF
			0:
				ATON1.PT := TIME_LAMP_TEST;
				ATON2.PT := TIME_LAMP_TEST;
				ATON3.PT := TIME_LAMP_TEST;
				gProgCamera.LED := 0;

				ATON1.IN := FALSE;
				IF (gMode = 1) AND ManualLampTest THEN
					gProgCamera.LED := 1;
					ManualLampTest := 0;
					ATON1.IN := TRUE;
					ATON2.IN := FALSE;
					sStep := 1;
				END_IF;

			1:
				gProgCamera.LED := 2;
				IF ATON1.Q THEN
					ATON2.IN := TRUE;
					ATON3.IN := FALSE;
					sStep := 2;
				END_IF;

			2:
				gProgCamera.LED := 3;
				IF ATON2.Q THEN
					sStep := 3;
				END_IF;

			3:
				gProgCamera.LED := 4;
				ATON3.IN := TRUE;
				ATON2.IN := FALSE;
				IF ATON3.Q THEN
					sStep := 0;
				END_IF;
		END_CASE;
	END_IF;

	//setting variable for recognised model with acknowledgement of 2 different types of B&R logos
	IF (gProgCamera.Model_ID=1) OR (gProgCamera.Model_ID=3) THEN
		gRecognisedModel := 1;
	ELSE
		gRecognisedModel := gProgCamera.Model_ID;
	END_IF

	//displaying last taken photo

	CASE ImageProcess OF	// state machine to process the picture to different destinations
		0:	// state to wait for commands and set next steps in process
			IF gProgCamera.DisplayPhoto THEN
				gProgCamera.DisplayPhoto := FALSE;
				ImageProcess := 1;
			END_IF

		1:	// get the image which is saved on the camera
			IF Logo.ModuleOK THEN
				ViBaseGetImage_0.MpLink := ADR(gCamera);
			ELSIF Color.ModuleOK THEN
				ViBaseGetImage_0.MpLink := ADR(gCamera_C);
			END_IF;
			ViBaseGetImage_0.Type := viBASE_IMAGE_TYPE_JPG;
			ViBaseGetImage_0.QualityLevel := VIBASE_GETIMG_QUALITY;
			ViBaseGetImage_0.Buffer := ADR(ViBaseBuffer);
			ViBaseGetImage_0.BufferSize := SIZEOF(ViBaseBuffer);
			ViBaseGetImage_0.Execute := TRUE;

			IF ViBaseGetImage_0.Error THEN
				ViBaseGetImage_0.Execute := FALSE;
				gProgCamera.DisplayPhoto := TRUE;
				ImageProcess := 0;
			END_IF;

			IF ViBaseGetImage_0.Done THEN
				Base64srcLen := ViBaseGetImage_0.BufferLen;	// save length of buffer on a local variable
				ViBaseGetImage_0.Execute := FALSE;

				ImageProcess := 2;
			END_IF

		2:	// transfer buffer to Base64 and merge the string to a valid SVG input
			IF NewEncodeReq THEN
				URL := '<image x=$'0$' y=$'0$' width=$'320px$' height=$'256px$' href=$'data:application/octet-stream;base64,';
				Base64Buffer := '';
				NewEncodeReq := FALSE;
			END_IF;

			httpEncodeBase64_0.pDest := ADR(Base64Buffer);
			httpEncodeBase64_0.destSize := SIZEOF(Base64Buffer) - strlen(ADR(Base64Buffer)) - strlen(ADR('$' />'));
			httpEncodeBase64_0.pSrc := ADR(ViBaseBuffer);
			httpEncodeBase64_0.srcLen := Base64srcLen;
			httpEncodeBase64_0.enable := TRUE;

			URLLength := strlen(ADR(URL));

			IF NOT(httpEncodeBase64_0.destLen=0) THEN
				gPhotoShowed := TRUE;
				strcat(ADR(Base64Buffer), ADR('$' />')) ; // Abschluss des Image Elements
				strcat(ADR(URL), ADR(Base64Buffer));

				NewEncodeReq := TRUE;
				URLLength := strlen(ADR(URL));
				httpEncodeBase64_0.enable := FALSE;

				ImageProcess := 0;
			END_IF;

	END_CASE;
	ViBaseGetImage_0();	// call FUB
	httpEncodeBase64_0();	// call FUB

END_PROGRAM

PROGRAM _EXIT

END_PROGRAM
```

### Program Logical/Programs/Alarms (IEC)

#### Variables.var
```iecst
VAR
	timerCycle : BOOL;
	redIconTimer : TON;
	pendingAlarms : BOOL;
	MpUserXConfig_0 : MpUserXConfig;
	MpUserXConfigType_0 : MpUserXConfigType;
	MpAlarmXHistory_0 : MpAlarmXHistory;
	MpAlarmXCore_0 : MpAlarmXCore;
	ModuleOkScale : BOOL;
	ModuleOkPneu_X67BC : BOOL;
	ModuleOkPLC_PLK : BOOL;
	ModuleOkInverter : BOOL;
	ModuleOkEncoder : BOOL;
	ModuleOkActuators : BOOL;
	isAcknowledged : BOOL;
	enableYellowIcon : BOOL;
	enableRedIcon : BOOL;
	ExportBool : BOOL;
	Export_Hist_Succ : BOOL;
END_VAR
```

#### Main.st
```iecst
PROGRAM _INIT
	(* Insert code here *)

END_PROGRAM

PROGRAM _CYCLIC

	MpAlarmXCore_0.Enable := TRUE;
	MpAlarmXCore_0.MpLink := ADR(gAlarmXCore);
	MpAlarmXCore_0();

	MpAlarmXHistory_0.Enable := TRUE;
	MpAlarmXHistory_0.MpLink := ADR(gAlarmXHistory);
	MpAlarmXHistory_0.DeviceName := ADR('CF_A');
	MpAlarmXHistory_0.Export := ExportBool;
	MpAlarmXHistory_0();

	MpUserXConfig_0.Enable := TRUE;
	MpUserXConfig_0.Configuration := ADR(MpUserXConfigType_0);
	MpUserXConfig_0();

	redIconTimer.PT := T#500ms;
	redIconTimer();

	// HARDWARE ALARM DETECTION
	IF NOT ModuleOkActuators OR NOT ModuleOkEncoder OR NOT ModuleOkInverter OR NOT ModuleOkPLC_PLK OR NOT ModuleOkPneu_X67BC OR NOT ModuleOkScale THEN
		gAlarmHardware := TRUE;
	ELSE
		gAlarmHardware := FALSE;
	END_IF;

	//isAcknowledged := MpAlarmXCheckState(gAlarmXCore, 'test_alarm', mpALARMX_STATE_ACKNOWLEDGED);
	IF (MpAlarmXCheckState(gAlarmXCore, 'Unrecognized object', mpALARMX_STATE_ACKNOWLEDGED) AND
		MpAlarmXCheckState(gAlarmXCore, 'Left box is full', mpALARMX_STATE_ACKNOWLEDGED) AND
		MpAlarmXCheckState(gAlarmXCore, 'Hardware error', mpALARMX_STATE_ACKNOWLEDGED) AND
		MpAlarmXCheckState(gAlarmXCore, 'Motor error', mpALARMX_STATE_ACKNOWLEDGED) AND
		MpAlarmXCheckState(gAlarmXCore, 'Right box is full', mpALARMX_STATE_ACKNOWLEDGED)) AND
		MpAlarmXCheckState(gAlarmXCore, 'Incorrect max left value', mpALARMX_STATE_ACKNOWLEDGED) AND
		MpAlarmXCheckState(gAlarmXCore, 'Incorrect min left value', mpALARMX_STATE_ACKNOWLEDGED) THEN
		isAcknowledged := TRUE;
	ELSE
		isAcknowledged := FALSE;
	END_IF;

	IF (MpAlarmXCore_0.PendingAlarms > 0) THEN
		pendingAlarms := TRUE;
	ELSE
		pendingAlarms := FALSE;
	END_IF;

	IF (MpAlarmXCore_0.ActiveAlarms = 0 AND MpAlarmXCore_0.PendingAlarms > 0) THEN
		enableYellowIcon := TRUE;
	ELSE
		enableYellowIcon := FALSE;
	END_IF;

	IF (MpAlarmXCore_0.ActiveAlarms > 0) THEN
		gAlarmExist := TRUE;
		IF (NOT(isAcknowledged)) THEN
			//blinking
			IF (redIconTimer.IN = FALSE) THEN
				redIconTimer.IN := TRUE;
			ELSIF (redIconTimer.Q) THEN
				timerCycle := NOT timerCycle;
				redIconTimer.IN := FALSE;
			END_IF;
			enableRedIcon := timerCycle;
		ELSE
			//static
			enableRedIcon := TRUE;
		END_IF;
	ELSE
		gAlarmExist := FALSE;
		enableRedIcon := FALSE;
	END_IF;

END_PROGRAM

PROGRAM _EXIT
	(* Insert code here *)

END_PROGRAM
```

### Program Logical/Programs/Program (ANSIC)

#### Main.cpp - Init, cyclic, exit code
```cpp
#include <bur/plctypes.h>

#ifdef _DEFAULT_INCLUDES
	#include <AsDefault.h>
#endif

// amount of memory to be allocated for heap storage must be specified for every ANSI C++ program with the bur_heap_size variable
unsigned long bur_heap_size = 0xFFFF;

void _INIT ProgramInit(void)
{
	// Insert code here

}

void _CYCLIC ProgramCyclic(void)
{
	// Insert code here

}

void _EXIT ProgramExit(void)
{
	// Insert code here

}
```

### Program Logical/Programs/SemiAuto

#### Types.typ
```iecst
TYPE
	ProgramStatesEnum :
		(
		STOP,
		INIT,
		DETECTION,
		CATEGORIZATION,
		SORT_STORAGE_LEFT,
		SORT_STORAGE_RIGHT,
		SORT_WEIGHT,
		SORT_WEIGHT_AND_OPTIC,
		SORT_OPTIC,
		STOP_AND_MANUAL,
		GO_STORAGE_LEFT,
		GO_STORAGE_RIGHT,
		TAKE_PICT_CAMERA,
		DROP,
		UNRECOGNISED_PIC,
		ERROR,
		START
	);
END_TYPE
```

#### Variables.var
```iecst
VAR
	Approval : BOOL;
	ActuatorByte : INT := 2#0000000000000000;
	ActuatorNotPushing : BOOL;
	ActuatorNotSorting : BOOL;
	ActuatorPushing : BOOL := FALSE;
	ActuatorSorting : BOOL := FALSE;
END_VAR
VAR CONSTANT
	ACTUATOR_BYTE_NOT_ACTIV : USINT := 2#0000000000000000;
	ACTUATOR_BYTE_PUSH : INT := 2#0000000000000100;
	ACTUATOR_BYTE_SORT : INT := 2#0000000000000001;
END_VAR
VAR
	IsEnglishSelected : BOOL := TRUE;
	ItemDetected : BOOL := FALSE;
	ItemWeight : USINT;
	ItemWeightMeasured : USINT;
	MotorHome : BOOL;
	MotorInPosition : BOOL;
	MotorMoveAbsolute : BOOL := FALSE;
	MotorMoveDone : BOOL;
	MotorPos : LREAL;
	MotorPower : BOOL := FALSE;
	MotorReqAcc : UINT := 700;
	MotorReqDec : UINT := 700;
	MotorReqPosition : UINT := 0;
	MotorReqVel : {REDUND_UNREPLICABLE} UINT := 300;
	MotorResetError : BOOL := FALSE;
	MotorVel : REAL;
END_VAR
VAR CONSTANT
	MOTOR_DIST_LEFT : UINT := 90;
	MOTOR_DIST_RIGHT : UINT := 320;
	RESET_ITEM_MEM_WEIGHT : USINT := 0;
END_VAR
VAR
	Start : BOOL := FALSE;
	State : ProgramStatesEnum := STOP;
	Stop : BOOL := FALSE;
	StringRecognisedModel : STRING[80];
	StringState : STRING[80];
	TimerActuatorOut : BOOL;
	TimerAfterDetect : BOOL;
	TimerCameraPicDone : BOOL;
	TimerTonActuator : TON;
	TimerTonActuatorIn : BOOL := FALSE;
	TimerTonCamera : TON;
	TimerTonDetect : TON;
END_VAR
VAR CONSTANT
	TIME_TON_ACTUATOR : TIME := T#500MS;
	TIME_TON_CAMERA : TIME := T#4S;
END_VAR
VAR
	TIME_TON_DETECT : TIME := T#2S;
	SemiAutoModeSelected : BOOL;
END_VAR
```

#### Main.st
```iecst
// ALREADY WORKING
PROGRAM _INIT
	// NEED ONLY FOR WATCH
	gAxis_1;
	gMotorBeltParType;
	gMotorBeltAxisBasic;
END_PROGRAM

PROGRAM _CYCLIC
	//CODE WORKS ONLY WHEN MANUAL MODE IS OFF
	SemiAutoModeSelected := (gMode=2);
	IF  SemiAutoModeSelected THEN

		// MOTOR MANAGEMENT
		gMotorBeltAxisBasic.Enable 		:= TRUE;
		gMotorBeltAxisBasic.MpLink 		:= ADR(gAxis_1);
		gMotorBeltAxisBasic.Parameters 	:= ADR(gMotorBeltParType);
		MotorMoveDone 					:= gMotorBeltAxisBasic.MoveDone;
		gMotorBeltAxisBasic.Power 		:= MotorPower;
		gMotorBeltAxisBasic.Home 		:= MotorHome;

		gMotorBeltAxisBasic();

		// IN STATE STOP VALUES DOESN'T FLUCTUATE
		IF gMotorBeltAxisBasic.Velocity > 15 THEN
			MotorVel := gMotorBeltAxisBasic.Velocity;
		ELSE
			MotorVel := 0;
		END_IF;
		IF gMotorBeltAxisBasic.Position > 5 THEN
			MotorPos := gMotorBeltAxisBasic.Position;
		ELSE
			MotorPos := 0;
		END_IF;

		// ASSIGNING MOTION PARAMETERS
		gMotorBeltParType.Acceleration 	:= MotorReqAcc;
		gMotorBeltParType.Deceleration 	:= MotorReqDec;
		gMotorBeltParType.Velocity 		:= MotorReqVel;
		gMotorBeltParType.Position 		:= MotorReqPosition;

		// ASSIGNING GLOBAL VARIABLES TO LOCAL VARIABLES
		gActuatorByte					 := ActuatorByte;
		gMotorBeltAxisBasic.Power 		 := MotorPower;
		gMotorBeltAxisBasic.MoveAbsolute := MotorMoveAbsolute;
		gStopState 						 := (State = 0);

		// ASSIGNING LOCAL VARIABLES TO GLOBAL VARIABLES
		MotorInPosition 				 := gMotorBeltAxisBasic.InPosition;
		ItemWeight 						 := gInWeightMeasure;

		// ITEM DETECTION CONDITION
		ItemDetected := (ItemWeight > 1);
		gWeightDetected := ItemDetected;

		// TIMERS
		// actuator
		TimerTonActuator(IN := TimerTonActuatorIn, PT := TIME_TON_ACTUATOR);
		TimerActuatorOut := TimerTonActuator.Q;
		// camera
		TimerTonCamera(IN := gProgCamera.ImageAcq , PT := TIME_TON_CAMERA);
		TimerCameraPicDone := TimerTonCamera.Q;
		// delay after detection
		TimerTonDetect.IN := ItemDetected;
		TimerTonDetect.PT := TIME_TON_DETECT;
		TimerAfterDetect := TimerTonDetect.Q;
		TimerTonDetect();
		// delay
		TimerTONShowPhoto.IN := gProgCamera.ImageAcq;
		TimerTONShowPhoto.PT := TIME_TON_SHOW_PHOTO;
		ShowPhoto := TimerTONShowPhoto.Q;
		TimerTONShowPhoto();

	END_IF;

	// ALARM OR STOP OR AUTO NOT ACTIVE
	IF	gAlarmHardware THEN
		IF NOT (State = ERROR) THEN
			State := ERROR;
		END_IF;
	ELSIF Stop OR gMode <> 0 OR gAlarmExist THEN
		Stop := FALSE;
		State := STOP;
	END_IF;

	// PROGRAM AUTO
	CASE State OF
		STOP:
			State := STOP;
			IF SemiAutoModeSelected THEN
				MotorPower 		  := FALSE;
				MotorMoveAbsolute := FALSE;
				MotorHome 		  := FALSE;
			END_IF;
			MotorPos := 0;
			MotorVel := 0;
			TimerTonActuatorIn 	  := FALSE;
			ActuatorSorting 	  := FALSE;
			ActuatorPushing  	  := FALSE;
			IF Start THEN
				State := INIT;
			END_IF;

		INIT:
			Sort_left			:= FALSE;
			Sort_right 			:= FALSE;
			gAddToRight 		:= FALSE;
			gAddToLeft 			:= FALSE;
			TimerTonActuatorIn 	:= FALSE;
			ActuatorSorting 	:= FALSE;
			ActuatorPushing 	:= FALSE;
			MotorMoveAbsolute 	:= FALSE;
			MotorPower 			:= TRUE;
			MotorHome 			:= TRUE;
			gPicNotRecognised	:= FALSE;
			State 				:= START;

		START:
			IF ItemDetected AND Approval THEN
				ItemWeightMeasured 	:= RESET_ITEM_MEM_WEIGHT;
				State := DETECTION;
			END_IF;

		DETECTION:
			MotorHome 	:= FALSE;
			IF TimerAfterDetect THEN
				ItemWeightMeasured := ItemWeight;
				State := CATEGORIZATION;
			END_IF;

		CATEGORIZATION:
			IF gSorting.SortChoice = WEIGHT THEN
				IF NOT gSorting.Threshold AND NOT (ItemWeightMeasured >= gSorting.ItemWeightLeftMin AND ItemWeightMeasured <= gSorting.ItemWeightLeftMax) AND NOT (ItemWeightMeasured >= gSorting.ItemWeightRightMin AND ItemWeightMeasured <= gSorting.ItemWeightRightMax) THEN
					State := UNRECOGNISED_PIC;//POTEM TO PRZENIES
				ELSE
					State := CHOOSE_SORT_MODE;
				END_IF;
			ELSE
				State := TAKE_PICT_CAMERA;
			END_IF;

		TAKE_PICT_CAMERA:
			StringState := 'Robienie zdjecia';
			gProgCamera.ImageAcq 	:= TRUE;
			IF TimerCameraPicDone AND Approval THEN
				gProgCamera.DisplayPhoto := TRUE;
				StringState := 'Zdjecie zrobione';
				Approval := 0;
				IF gRecognisedModel = 0 THEN 						//0
					gProgCamera.ImageAcq 			  := FALSE;
					StringRecognisedModel := 'Unrecognised';
					State 				  := UNRECOGNISED_PIC;
				ELSE
					State 				  := DROP;
				END_IF;
			END_IF;

		DROP:
			StringState := 'Dozowanie detalu';
			ActuatorPushing := TRUE;
			IF TimerActuatorOut THEN
				ActuatorPushing := FALSE;
				IF gSorting.SortChoice = OPTIC_LOGO OR gSorting.SortChoice = OPTIC_COLOR THEN
					gSortChoiceView := TRUE;
					State := SORT_OPTIC;
				ELSIF gSorting.SortChoice = WEIGHT THEN
					gSortChoiceView := FALSE;
					State := SORT_WEIGHT;
				END_IF;
			END_IF;

		// ABOVE 1 TO ItemWeightChoosen ITEM FALL INTO THE LEFT, EQUAL AND ABOVE ItemWeightChoosen INTO THE RIGHT
		SORT_WEIGHT:
			IF (ItemWeightMeasured >= gSorting.ItemWeightLeftMin AND ItemWeightMeasured < gSorting.ItemWeightLeftMax) AND NOT (ItemWeightMeasured >= gSorting.ItemWeightRightMin AND ItemWeightMeasured < gSorting.ItemWeightRightMax)  THEN
				IF gSorting.SortLeftMin THEN
					State := GO_STORAGE_LEFT;
				ELSE
					State := GO_STORAGE_RIGHT;
				END_IF;
			ELSIF (ItemWeightMeasured >= gSorting.ItemWeightRightMin AND ItemWeightMeasured < gSorting.ItemWeightRightMax) AND NOT (ItemWeightMeasured >= gSorting.ItemWeightLeftMin AND ItemWeightMeasured < gSorting.ItemWeightLeftMax) THEN
				IF gSorting.SortLeftMin THEN
					State := GO_STORAGE_RIGHT;
				ELSE
					State := GO_STORAGE_LEFT;
				END_IF;
			ELSE
				State := ERROR;
				//ALARM
			END_IF;

		SORT_OPTIC:
			StringState := 'Sortowanie optyczne';
			IF gRecognisedModel = 1 THEN
				gProgCamera.ImageAcq 			  := FALSE;
				StringRecognisedModel := 'B&R';					//1
				IF gSorting.SortLeftBR AND Approval THEN
					Approval := 0;
					State := GO_STORAGE_LEFT;
				ELSE
					IF Approval THEN
						Approval := 0;
						State := GO_STORAGE_RIGHT;
					END_IF;
				END_IF;

			ELSIF gRecognisedModel = 2 THEN						//2
				gProgCamera.ImageAcq 			  := FALSE;
				StringRecognisedModel := 'AS';
				IF gSorting.SortLeftBR AND Approval THEN
					Approval := 0;
					State := GO_STORAGE_RIGHT;
				ELSE
					IF Approval THEN
						Approval := 0;
						State := GO_STORAGE_LEFT;
					END_IF;
				END_IF;
			END_IF;

		GO_STORAGE_LEFT:
			StringState := 'Transport detalu do lewego zbiornika';
			MotorReqPosition := MOTOR_DIST_LEFT;
			MotorMoveAbsolute := TRUE;
			IF MotorInPosition AND MotorMoveDone AND Approval THEN
				Approval := 0;
				State := SORT_STORAGE_LEFT;
			END_IF;

		GO_STORAGE_RIGHT:
			StringState := 'Transport detalu do prawego zbiornika';
			MotorReqPosition  := MOTOR_DIST_RIGHT;
			MotorMoveAbsolute := TRUE;
			IF MotorInPosition AND MotorMoveDone AND Approval THEN
				Approval := 0;
				State := SORT_STORAGE_RIGHT;
			END_IF;

		SORT_STORAGE_LEFT:
			StringState := 'Zepchniecie detalu z tasmy do zbiornika lewego';
			MotorMoveAbsolute := FALSE;
			ActuatorSorting   := TRUE;
			gAddToLeft 		  := TRUE;
			IF TimerActuatorOut THEN
				State := INIT;
			END_IF;

		SORT_STORAGE_RIGHT:
			gAddToRight := TRUE;
			MotorMoveAbsolute := FALSE;
			State := INIT;

		UNRECOGNISED_PIC:
			StringState := 'Nie rozpoznano zdjecia';
			gPicNotRecognised := TRUE;
			State := STOP;

		ERROR:
			StringState := 'Wystapil blad';
			gErrorState := TRUE;
			IF gAlarmHardAck THEN
				IF NOT gAlarmHardware THEN
					gAlarmHardAck := FALSE;
					gErrorState := FALSE;
					State := STOP;
				END_IF;
			END_IF;

	END_CASE;

	// TIMER INPUT TRIGGER TO DELAY ACTUATORS
	IF ActuatorPushing OR ActuatorSorting THEN
		TimerTonActuatorIn := TRUE;
	ELSE
		TimerTonActuatorIn := FALSE;
	END_IF;

	// OPERATION OF BYTE ACTUATORS WITH TIMER
	IF ActuatorPushing THEN
		ActuatorByte := ACTUATOR_BYTE_PUSH;
		IF TimerActuatorOut THEN
			ActuatorPushing := FALSE;
		END_IF;
	ELSIF ActuatorSorting THEN
		ActuatorByte := ACTUATOR_BYTE_SORT;
		IF TimerActuatorOut THEN
			ActuatorSorting := FALSE;
		END_IF;
	ELSE
		ActuatorByte := ACTUATOR_BYTE_NOT_ACTIV;
	END_IF;

	// HMI GUYS WANTED SOME VARIABLES
	IF gSorting.SortChoice = OPTIC_LOGO OR gSorting.SortChoice = OPTIC_COLOR THEN
		gSortChoiceView := TRUE;
	ELSIF gSorting.SortChoice = WEIGHT THEN
		gSortChoiceView := FALSE;
	END_IF;

	ActuatorNotSorting := NOT ActuatorSorting;
	ActuatorNotPushing 	:= NOT ActuatorPushing;

	IF Start THEN
		Start := FALSE;
	END_IF;

	//Added by Jakub; Responsibler for changing machine state between English and Polish
	IF IsEnglishSelected THEN
		IF StringState = 'Inicjalizacja' THEN
			StringState := 'Initialization';

		ELSIF StringState = 'Zdjecie zrobione' THEN
			StringState := 'Picture taken';

		ELSIF StringState = 'Gotowy do startu' THEN
			StringState := 'Ready';

		ELSIF StringState = 'Wykrycie detalu' THEN
			StringState := 'Item detection';

		ELSIF StringState = 'Kategoryzacja detalu' THEN
			StringState := 'Item categorization';

		ELSIF StringState = 'Robienie zdjecia' THEN
			StringState := 'Taking a picture';

		ELSIF StringState = 'Dozowanie detalu' THEN
			StringState := 'Item dosing';

		ELSIF StringState = 'Sortowanie wagowe' THEN
			StringState := 'Sorting by weight';

		ELSIF StringState = 'Sortowanie optyczne' THEN
			StringState := 'Optical sorting';

		ELSIF StringState = 'Transport detalu do lewego zbiornika' THEN
			StringState := 'Item transport to the left tank';

		ELSIF StringState = 'Transport detalu do prawego zbiornika' THEN
			StringState := 'Item transport to the right tank';

		ELSIF StringState = 'Zepchniecie detalu z tasmy do zbiornika lewego' THEN
			StringState := 'Pushing the item from the belt to the left tank';

		ELSIF StringState = 'Nie rozpoznano zdjecia' THEN
			StringState := 'Photo not recognized';

		ELSIF StringState = 'Stop' THEN
			StringState := 'Stop';

		ELSIF StringState = 'Wystapil blad' THEN
			StringState := 'Error';

		ELSIF StringState = 'Gotowy do startu' THEN
			StringState := 'Ready to start';
		END_IF;
	END_IF;

		END_PROGRAM

PROGRAM _EXIT

		END_PROGRAM
```

- Project.language (not shown)

- Sorter POWERLINK.pptx (binary file, 1488936 bytes)
Listed in the project but not available here: Logical/Programs/Program/Types.typ, Logical/Programs/Program/Variables.var
